KUKA KRL program: EPS_2_25862_MH6A_A_20251016034303.src

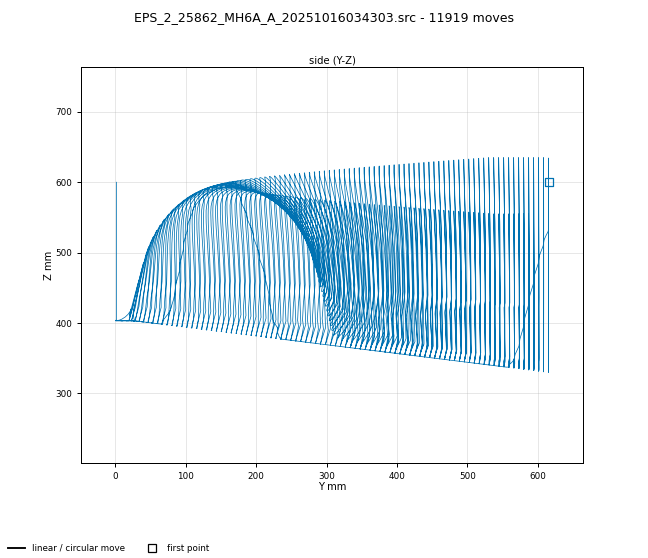
[picture p0: tool path of EPS_2_25862_MH6A_A_20251016034303.src, 11919 of 11921 moves have a stored position in this frame; points joined in program order, loops and branches not executed]
&ACCESS RVP
&REL 4
&COMMENT QRS 19112012
&PARAM EDITMASK = *
DEF PART()
EXT BAS (BAS_COMMAND :IN,REAL :IN )
INT I
BAS (#INITMOV,0 )

;KUKA QRS Post kuka4.cps  Date:22-06-2017 !

File_ID=2890

QRS_PRE_INIT()

;Init var - Until changes are made in qrs_pre_init
Outlet_Square_prg=0
Inlet_1_Square_prg=0
Inlet_2_Square_prg=0
Inlet_3_Square_prg=0
Inlet_4_Square_prg=0
Inlet_5_Square_prg=0

Outlet_1={X 0.000, Y 530.070, Z 534.500, B 0.000, E1 0.000 }
Inlet_1={X 0.000, Y 535.780, Z 454.500, B 0.000, E1 90.000 }
Outlet_1_type=201
Inlet_1_type=201
;QRS#1=Sidecore dimensions
;QRS#2=200-8" PVC SDR 35
;QRS#3=200-8" PVC SDR 35
;QRS#4=
;QRS#5=
;QRS#6=
;QRS#7=
;QRS#8=
;QRS#9=12-08 PSX
;QRS#10=12-08 PSX
;QRS#11=
;QRS#12=
;QRS#13=
;QRS#14=
;QRS#15=
;QRS#16=1220x127x914 3'
;QRS#17=EPS Height
;QRS#18=635
;QRS#19=*
;QRS#20= UPDATED VERSION 22-06-2017
;QRS#21=*
Outlet_Square=0100
Inlet_1_Square=0100
Inlet_2_Square=0
Inlet_3_Square=0
Inlet_4_Square=0
Inlet_5_Square=0
Mill_Square=1
Outlet_Square_Prg=204
Inlet_1_Square_prg=204

QRS_INIT()

$ADVANCE=5

; T1
PTP {E1 173.497,E2 173.497}
PTP {X 0,Y 615.499,A -85,B 0,C 180,E1 173.497,E2 173.497,E3 0,E4 0,E5 0,E6 0}
QRS_SPEED_INIT()
LIN {X 0,Y 615.499,Z 600,A -85,B 0,C 180,E1 173.497,E2 173.497,E3 0,E4 0,E5 0,E6 0} C_VEL
LIN {X 0,Y 615.499,Z 545.726,A -85,B 0,C 180,E1 173.497,E2 173.497} C_VEL
LIN {X 0,Y 615.499,Z 534.845,A -85,B 0,C 180,E1 173.497,E2 173.497} C_VEL
LIN {X 0,Y 615.497,Z 533.201,A -85,B 0,C 180,E1 173.417,E2 173.417} C_VEL
LIN {X 0,Y 615.497,Z 525.537,A -85,B 0,C 180,E1 172.455,E2 172.455} C_VEL
LIN {X 0,Y 615.498,Z 515.759,A -85,B 0,C 180,E1 171.464,E2 171.464} C_VEL
LIN {X 0,Y 615.497,Z 505.494,A -85,B 0,C 180,E1 170.636,E2 170.636} C_VEL
LIN {X 0,Y 615.479,Z 493.933,A -85,B 0,C 180,E1 169.889,E2 169.889} C_VEL
LIN {X 0,Y 615.498,Z 482.051,A -85,B 0,C 180,E1 169.292,E2 169.292} C_VEL
LIN {X 0,Y 615.49,Z 469.16,A -85,B 0,C 180,E1 168.807,E2 168.807} C_VEL
LIN {X 0,Y 615.493,Z 456.56,A -85,B 0,C 180,E1 168.473,E2 168.473} C_VEL
LIN {X 0,Y 615.494,Z 443.437,A -85,B 0,C 180,E1 168.265,E2 168.265} C_VEL
LIN {X 0,Y 615.492,Z 345.168,A -85,B 0,C 180,E1 167.114,E2 167.114} C_VEL
LIN {X 0,Y 615.479,Z 330.504,A -85,B 0,C 180,E1 164.265,E2 164.265} C_VEL
LIN {X 0,Y 615.477,Z 329.689,A -85,B 0,C 180,E1 164.095,E2 164.095} C_VEL
LIN {X 0,Y 615.484,Z 329.685,A -85,B 0,C 180,E1 161.354,E2 161.354} C_VEL
LIN {X 0,Y 615.494,Z 329.697,A -85,B 0,C 180,E1 158.568,E2 158.568} C_VEL
LIN {X 0,Y 615.488,Z 329.682,A -85,B 0,C 180,E1 155.728,E2 155.728} C_VEL
LIN {X 0,Y 615.488,Z 329.7,A -85,B 0,C 180,E1 152.823,E2 152.823} C_VEL
LIN {X 0,Y 615.477,Z 329.688,A -85,B 0,C 180,E1 150.208,E2 150.208} C_VEL
LIN {X 0,Y 615.491,Z 329.683,A -85,B 0,C 180,E1 147.543,E2 147.543} C_VEL
LIN {X 0,Y 615.483,Z 329.692,A -85,B 0,C 180,E1 145.185,E2 145.185} C_VEL
LIN {X 0,Y 615.495,Z 329.697,A -85,B 0,C 180,E1 142.758,E2 142.758} C_VEL
LIN {X 0,Y 615.486,Z 329.683,A -85,B 0,C 180,E1 139.912,E2 139.912} C_VEL
LIN {X 0,Y 615.494,Z 329.682,A -85,B 0,C 180,E1 137.648,E2 137.648} C_VEL
LIN {X 0,Y 615.497,Z 329.7,A -85,B 0,C 180,E1 134.932,E2 134.932} C_VEL
LIN {X 0,Y 615.479,Z 329.684,A -85,B 0,C 180,E1 132.079,E2 132.079} C_VEL
LIN {X 0,Y 615.495,Z 329.682,A -85,B 0,C 180,E1 129.75,E2 129.75} C_VEL
LIN {X 0,Y 615.494,Z 329.697,A -85,B 0,C 180,E1 126.937,E2 126.937} C_VEL
LIN {X 0,Y 615.482,Z 329.683,A -85,B 0,C 180,E1 124.023,E2 124.023} C_VEL
LIN {X 0,Y 615.492,Z 329.701,A -85,B 0,C 180,E1 121.086,E2 121.086} C_VEL
LIN {X 0,Y 615.477,Z 329.686,A -85,B 0,C 180,E1 118.448,E2 118.448} C_VEL
LIN {X 0,Y 615.493,Z 329.685,A -85,B 0,C 180,E1 115.716,E2 115.716} C_VEL
LIN {X 0,Y 615.49,Z 329.69,A -85,B 0,C 180,E1 112.845,E2 112.845} C_VEL
LIN {X 0,Y 615.483,Z 329.684,A -85,B 0,C 180,E1 110.034,E2 110.034} C_VEL
LIN {X 0,Y 615.497,Z 329.701,A -85,B 0,C 180,E1 107.271,E2 107.271} C_VEL
LIN {X 0,Y 615.479,Z 329.686,A -85,B 0,C 180,E1 104.55,E2 104.55} C_VEL
LIN {X 0,Y 615.49,Z 329.686,A -85,B 0,C 180,E1 101.861,E2 101.861} C_VEL
LIN {X 0,Y 615.496,Z 329.695,A -85,B 0,C 180,E1 99.199,E2 99.199} C_VEL
LIN {X 0,Y 615.478,Z 329.685,A -85,B 0,C 180,E1 96.557,E2 96.557} C_VEL
LIN {X 0,Y 615.491,Z 329.686,A -85,B 0,C 180,E1 93.929,E2 93.929} C_VEL
LIN {X 0,Y 615.496,Z 329.696,A -85,B 0,C 180,E1 91.309,E2 91.309} C_VEL
LIN {X 0,Y 615.48,Z 329.685,A -85,B 0,C 180,E1 88.692,E2 88.692} C_VEL
LIN {X 0,Y 615.489,Z 329.686,A -85,B 0,C 180,E1 86.072,E2 86.072} C_VEL
LIN {X 0,Y 615.496,Z 329.696,A -85,B 0,C 180,E1 83.416,E2 83.416} C_VEL
LIN {X 0,Y 615.48,Z 329.685,A -85,B 0,C 180,E1 80.802,E2 80.802} C_VEL
LIN {X 0,Y 615.488,Z 329.687,A -85,B 0,C 180,E1 78.14,E2 78.14} C_VEL
LIN {X 0,Y 615.494,Z 329.695,A -85,B 0,C 180,E1 75.452,E2 75.452} C_VEL
LIN {X 0,Y 615.478,Z 329.685,A -85,B 0,C 180,E1 72.73,E2 72.73} C_VEL
LIN {X 0,Y 615.494,Z 329.692,A -85,B 0,C 180,E1 69.968,E2 69.968} C_VEL
LIN {X 0,Y 615.49,Z 329.686,A -85,B 0,C 180,E1 67.157,E2 67.157} C_VEL
LIN {X 0,Y 615.489,Z 329.686,A -85,B 0,C 180,E1 64.285,E2 64.285} C_VEL
LIN {X 0,Y 615.491,Z 329.688,A -85,B 0,C 180,E1 61.343,E2 61.343} C_VEL
LIN {X 0,Y 615.482,Z 329.684,A -85,B 0,C 180,E1 58.915,E2 58.915} C_VEL
LIN {X 0,Y 615.482,Z 329.686,A -85,B 0,C 180,E1 56.467,E2 56.467} C_VEL
LIN {X 0,Y 615.493,Z 329.691,A -85,B 0,C 180,E1 54.166,E2 54.166} C_VEL
LIN {X 0,Y 615.496,Z 329.699,A -85,B 0,C 180,E1 51.933,E2 51.933} C_VEL
LIN {X 0,Y 615.487,Z 329.687,A -85,B 0,C 180,E1 49.395,E2 49.395} C_VEL
LIN {X 0,Y 615.476,Z 329.685,A -85,B 0,C 180,E1 46.756,E2 46.756} C_VEL
LIN {X 0,Y 615.491,Z 329.701,A -85,B 0,C 180,E1 43.999,E2 43.999} C_VEL
LIN {X 0,Y 615.49,Z 329.686,A -85,B 0,C 180,E1 41.474,E2 41.474} C_VEL
LIN {X 0,Y 615.478,Z 329.685,A -85,B 0,C 180,E1 38.905,E2 38.905} C_VEL
LIN {X 0,Y 615.488,Z 329.691,A -85,B 0,C 180,E1 36.425,E2 36.425} C_VEL
LIN {X 0,Y 615.489,Z 329.686,A -85,B 0,C 180,E1 33.536,E2 33.536} C_VEL
LIN {X 0,Y 615.478,Z 329.685,A -85,B 0,C 180,E1 30.92,E2 30.92} C_VEL
LIN {X 0,Y 615.491,Z 329.692,A -85,B 0,C 180,E1 28.453,E2 28.453} C_VEL
LIN {X 0,Y 615.488,Z 329.685,A -85,B 0,C 180,E1 25.572,E2 25.572} C_VEL
LIN {X 0,Y 615.475,Z 329.688,A -85,B 0,C 180,E1 22.845,E2 22.845} C_VEL
LIN {X 0,Y 615.487,Z 329.695,A -85,B 0,C 180,E1 20.033,E2 20.033} C_VEL
LIN {X 0,Y 615.489,Z 329.682,A -85,B 0,C 180,E1 17.27,E2 17.27} C_VEL
LIN {X 0,Y 615.49,Z 329.694,A -85,B 0,C 180,E1 14.549,E2 14.549} C_VEL
LIN {X 0,Y 615.481,Z 329.689,A -85,B 0,C 180,E1 11.861,E2 11.861} C_VEL
LIN {X 0,Y 615.483,Z 329.684,A -85,B 0,C 180,E1 9.199,E2 9.199} C_VEL
LIN {X 0,Y 615.492,Z 329.696,A -85,B 0,C 180,E1 6.557,E2 6.557} C_VEL
LIN {X 0,Y 615.476,Z 329.69,A -85,B 0,C 180,E1 3.929,E2 3.929} C_VEL
LIN {X 0,Y 615.486,Z 329.683,A -85,B 0,C 180,E1 1.309,E2 1.309} C_VEL
LIN {X 0,Y 615.485,Z 329.696,A -85,B 0,C 180,E1 -1.309,E2 -1.309} C_VEL
LIN {X 0,Y 615.476,Z 329.691,A -85,B 0,C 180,E1 -3.929,E2 -3.929} C_VEL
LIN {X 0,Y 615.49,Z 329.682,A -85,B 0,C 180,E1 -6.59,E2 -6.59} C_VEL
LIN {X 0,Y 615.483,Z 329.696,A -85,B 0,C 180,E1 -9.199,E2 -9.199} C_VEL
LIN {X 0,Y 615.478,Z 329.69,A -85,B 0,C 180,E1 -11.861,E2 -11.861} C_VEL
LIN {X 0,Y 615.49,Z 329.682,A -85,B 0,C 180,E1 -14.549,E2 -14.549} C_VEL
LIN {X 0,Y 615.495,Z 329.699,A -85,B 0,C 180,E1 -17.27,E2 -17.27} C_VEL
LIN {X 0,Y 615.479,Z 329.686,A -85,B 0,C 180,E1 -20.033,E2 -20.033} C_VEL
LIN {X 0,Y 615.482,Z 329.69,A -85,B 0,C 180,E1 -22.845,E2 -22.845} C_VEL
LIN {X 0,Y 615.485,Z 329.692,A -85,B 0,C 180,E1 -25.571,E2 -25.571} C_VEL
LIN {X 0,Y 615.492,Z 329.682,A -85,B 0,C 180,E1 -28.454,E2 -28.454} C_VEL
LIN {X 0,Y 615.487,Z 329.7,A -85,B 0,C 180,E1 -31.088,E2 -31.088} C_VEL
LIN {X 0,Y 615.484,Z 329.691,A -85,B 0,C 180,E1 -33.536,E2 -33.536} C_VEL
LIN {X 0,Y 615.489,Z 329.684,A -85,B 0,C 180,E1 -36.425,E2 -36.425} C_VEL
LIN {X 0,Y 615.496,Z 329.7,A -85,B 0,C 180,E1 -39.065,E2 -39.065} C_VEL
LIN {X 0,Y 615.485,Z 329.69,A -85,B 0,C 180,E1 -41.474,E2 -41.474} C_VEL
LIN {X 0,Y 615.491,Z 329.682,A -85,B 0,C 180,E1 -44.149,E2 -44.149} C_VEL
LIN {X 0,Y 615.492,Z 329.7,A -85,B 0,C 180,E1 -46.952,E2 -46.952} C_VEL
LIN {X 0,Y 615.483,Z 329.69,A -85,B 0,C 180,E1 -49.395,E2 -49.395} C_VEL
LIN {X 0,Y 615.484,Z 329.683,A -85,B 0,C 180,E1 -51.989,E2 -51.989} C_VEL
LIN {X 0,Y 615.491,Z 329.686,A -85,B 0,C 180,E1 -54.386,E2 -54.386} C_VEL
LIN {X 0,Y 615.487,Z 329.698,A -85,B 0,C 180,E1 -56.765,E2 -56.765} C_VEL
LIN {X 0,Y 615.496,Z 329.693,A -85,B 0,C 180,E1 -59.082,E2 -59.082} C_VEL
LIN {X 0,Y 615.477,Z 329.686,A -85,B 0,C 180,E1 -61.552,E2 -61.552} C_VEL
LIN {X 0,Y 615.493,Z 329.686,A -85,B 0,C 180,E1 -64.286,E2 -64.286} C_VEL
LIN {X 0,Y 615.483,Z 329.765,A -85,B 0,C 180,E1 -66.022,E2 -66.022} C_VEL
LIN {X 0,Y 615.486,Z 351.817,A -85,B 0,C 180,E1 -68.745,E2 -68.745} C_VEL
LIN {X 0,Y 615.494,Z 375,A -85,B 0,C 180,E1 -71.556,E2 -71.556} C_VEL
LIN {X 0,Y 615.486,Z 397.682,A -85,B 0,C 180,E1 -74.266,E2 -74.266} C_VEL
LIN {X 0,Y 615.498,Z 421.822,A -85,B 0,C 180,E1 -77.115,E2 -77.115} C_VEL
LIN {X 0,Y 615.479,Z 530.88,A -85,B 0,C 180,E1 -78.411,E2 -78.411} C_VEL
LIN {X 0,Y 615.478,Z 543.377,A -85,B 0,C 180,E1 -78.683,E2 -78.683} C_VEL
LIN {X 0,Y 615.491,Z 556.57,A -85,B 0,C 180,E1 -79.111,E2 -79.111} C_VEL
LIN {X 0,Y 615.478,Z 568.495,A -85,B 0,C 180,E1 -79.64,E2 -79.64} C_VEL
LIN {X 0,Y 615.487,Z 580.008,A -85,B 0,C 180,E1 -80.305,E2 -80.305} C_VEL
LIN {X 0,Y 615.499,Z 590.352,A -85,B 0,C 180,E1 -81.051,E2 -81.051} C_VEL
LIN {X 0,Y 615.497,Z 598.82,A -85,B 0,C 180,E1 -81.795,E2 -81.795} C_VEL
LIN {X 0,Y 615.497,Z 607.972,A -85,B 0,C 180,E1 -82.785,E2 -82.785} C_VEL
LIN {X 0,Y 615.497,Z 615.321,A -85,B 0,C 180,E1 -83.773,E2 -83.773} C_VEL
LIN {X 0,Y 615.499,Z 621.209,A -85,B 0,C 180,E1 -84.76,E2 -84.76} C_VEL
LIN {X 0,Y 615.493,Z 625.855,A -85,B 0,C 180,E1 -85.744,E2 -85.744} C_VEL
LIN {X 0,Y 615.495,Z 629.401,A -85,B 0,C 180,E1 -86.728,E2 -86.728} C_VEL
LIN {X 0,Y 615.497,Z 631.235,A -85,B 0,C 180,E1 -87.383,E2 -87.383} C_VEL
LIN {X 0,Y 615.497,Z 632.609,A -85,B 0,C 180,E1 -88.038,E2 -88.038} C_VEL
LIN {X 0,Y 615.496,Z 634.174,A -85,B 0,C 180,E1 -89.347,E2 -89.347} C_VEL
LIN {X 0,Y 615.494,Z 634.389,A -85,B 0,C 180,E1 -90.001,E2 -90.001} C_VEL
LIN {X 0,Y 615.496,Z 633.579,A -85,B 0,C 180,E1 -91.309,E2 -91.309} C_VEL
LIN {X 0,Y 615.497,Z 632.607,A -85,B 0,C 180,E1 -91.964,E2 -91.964} C_VEL
LIN {X 0,Y 615.497,Z 631.231,A -85,B 0,C 180,E1 -92.619,E2 -92.619} C_VEL
LIN {X 0,Y 615.496,Z 628.347,A -85,B 0,C 180,E1 -93.601,E2 -93.601} C_VEL
LIN {X 0,Y 615.498,Z 624.438,A -85,B 0,C 180,E1 -94.585,E2 -94.585} C_VEL
LIN {X 0,Y 615.499,Z 619.401,A -85,B 0,C 180,E1 -95.57,E2 -95.57} C_VEL
LIN {X 0,Y 615.497,Z 612.87,A -85,B 0,C 180,E1 -96.583,E2 -96.583} C_VEL
LIN {X 0,Y 615.497,Z 605.127,A -85,B 0,C 180,E1 -97.546,E2 -97.546} C_VEL
LIN {X 0,Y 615.498,Z 597.037,A -85,B 0,C 180,E1 -98.372,E2 -98.372} C_VEL
LIN {X 0,Y 615.499,Z 587.158,A -85,B 0,C 180,E1 -99.199,E2 -99.199} C_VEL
LIN {X 0,Y 615.488,Z 575.97,A -85,B 0,C 180,E1 -99.946,E2 -99.946} C_VEL
LIN {X 0,Y 615.481,Z 565.009,A -85,B 0,C 180,E1 -100.528,E2 -100.528} C_VEL
LIN {X 0,Y 615.49,Z 552.439,A -85,B 0,C 180,E1 -101.042,E2 -101.042} C_VEL
LIN {X 0,Y 615.477,Z 540.037,A -85,B 0,C 180,E1 -101.402,E2 -101.402} C_VEL
LIN {X 0,Y 615.481,Z 526.418,A -85,B 0,C 180,E1 -101.653,E2 -101.653} C_VEL
LIN {X 0,Y 615.498,Z 421.809,A -85,B 0,C 180,E1 -102.887,E2 -102.887} C_VEL
LIN {X 0,Y 615.486,Z 397.669,A -85,B 0,C 180,E1 -105.736,E2 -105.736} C_VEL
LIN {X 0,Y 615.498,Z 373.644,A -85,B 0,C 180,E1 -108.607,E2 -108.607} C_VEL
LIN {X 0,Y 615.488,Z 350.368,A -85,B 0,C 180,E1 -111.432,E2 -111.432} C_VEL
LIN {X 0,Y 615.486,Z 329.684,A -85,B 0,C 180,E1 -114.007,E2 -114.007} C_VEL
LIN {X 0,Y 615.478,Z 329.686,A -85,B 0,C 180,E1 -116.445,E2 -116.445} C_VEL
LIN {X 0,Y 615.485,Z 329.688,A -85,B 0,C 180,E1 -118.659,E2 -118.659} C_VEL
LIN {X 0,Y 615.495,Z 329.699,A -85,B 0,C 180,E1 -121.087,E2 -121.087} C_VEL
LIN {X 0,Y 615.483,Z 329.683,A -85,B 0,C 180,E1 -124.023,E2 -124.023} C_VEL
LIN {X 0,Y 615.494,Z 329.696,A -85,B 0,C 180,E1 -126.937,E2 -126.937} C_VEL
LIN {X 0,Y 615.495,Z 329.682,A -85,B 0,C 180,E1 -129.75,E2 -129.75} C_VEL
LIN {X 0,Y 615.476,Z 329.687,A -85,B 0,C 180,E1 -132.355,E2 -132.355} C_VEL
LIN {X 0,Y 615.493,Z 329.699,A -85,B 0,C 180,E1 -135.069,E2 -135.069} C_VEL
LIN {X 0,Y 615.486,Z 329.683,A -85,B 0,C 180,E1 -137.921,E2 -137.921} C_VEL
LIN {X 0,Y 615.477,Z 329.686,A -85,B 0,C 180,E1 -140.249,E2 -140.249} C_VEL
LIN {X 0,Y 615.492,Z 329.697,A -85,B 0,C 180,E1 -143.064,E2 -143.064} C_VEL
LIN {X 0,Y 615.481,Z 329.684,A -85,B 0,C 180,E1 -145.977,E2 -145.977} C_VEL
LIN {X 0,Y 615.479,Z 329.688,A -85,B 0,C 180,E1 -148.314,E2 -148.314} C_VEL
LIN {X 0,Y 615.489,Z 329.693,A -85,B 0,C 180,E1 -150.594,E2 -150.594} C_VEL
LIN {X 0,Y 615.494,Z 329.682,A -85,B 0,C 180,E1 -153.556,E2 -153.556} C_VEL
LIN {X 0,Y 615.485,Z 329.691,A -85,B 0,C 180,E1 -156.443,E2 -156.443} C_VEL
LIN {X 0,Y 615.484,Z 329.688,A -85,B 0,C 180,E1 -159.269,E2 -159.269} C_VEL
LIN {X 0,Y 615.477,Z 329.686,A -85,B 0,C 180,E1 -162.043,E2 -162.043} C_VEL
LIN {X 0,Y 615.478,Z 329.826,A -85,B 0,C 180,E1 -164.222,E2 -164.222} C_VEL
LIN {X 0,Y 615.495,Z 343.07,A -85,B 0,C 180,E1 -166.799,E2 -166.799} C_VEL
LIN {X 0,Y 615.494,Z 345.135,A -85,B 0,C 180,E1 -167.197,E2 -167.197} C_VEL
LIN {X 0,Y 615.494,Z 450.636,A -85,B 0,C 180,E1 -168.452,E2 -168.452} C_VEL
LIN {X 0,Y 615.491,Z 463.219,A -85,B 0,C 180,E1 -168.724,E2 -168.724} C_VEL
LIN {X 0,Y 615.491,Z 476.604,A -85,B 0,C 180,E1 -169.158,E2 -169.158} C_VEL
LIN {X 0,Y 615.492,Z 487.563,A -85,B 0,C 180,E1 -169.639,E2 -169.639} C_VEL
LIN {X 0,Y 615.482,Z 499.304,A -85,B 0,C 180,E1 -170.304,E2 -170.304} C_VEL
LIN {X 0,Y 615.499,Z 509.766,A -85,B 0,C 180,E1 -171.05,E2 -171.05} C_VEL
LIN {X 0,Y 615.498,Z 518.329,A -85,B 0,C 180,E1 -171.794,E2 -171.794} C_VEL
LIN {X 0,Y 615.498,Z 526.208,A -85,B 0,C 180,E1 -172.619,E2 -172.619} C_VEL
LIN {X 0,Y 615.497,Z 533.898,A -85,B 0,C 180,E1 -173.608,E2 -173.608} C_VEL
LIN {X 0,Y 615.498,Z 540.957,A -85,B 0,C 180,E1 -174.759,E2 -174.759} C_VEL
LIN {X 0,Y 615.493,Z 545.657,A -85,B 0,C 180,E1 -175.744,E2 -175.744} C_VEL
LIN {X 0,Y 615.496,Z 549.254,A -85,B 0,C 180,E1 -176.727,E2 -176.727} C_VEL
LIN {X 0,Y 615.496,Z 551.114,A -85,B 0,C 180,E1 -177.382,E2 -177.382} C_VEL
LIN {X 0,Y 615.497,Z 552.533,A -85,B 0,C 180,E1 -178.037,E2 -178.037} C_VEL
LIN {X 0,Y 615.496,Z 554.141,A -85,B 0,C 180,E1 -179.346,E2 -179.346} C_VEL
LIN {X 0,Y 615.494,Z 554.384,A -85,B 0,C 180,E1 -180,E2 -180} C_VEL
LIN {X 0,Y 615.496,Z 554.206,A -85,B 0,C 180,E1 -180.654,E2 -180.654} C_VEL
LIN {X 0,Y 615.496,Z 552.683,A -85,B 0,C 180,E1 -181.963,E2 -181.963} C_VEL
LIN {X 0,Y 615.498,Z 551.341,A -85,B 0,C 180,E1 -182.618,E2 -182.618} C_VEL
LIN {X 0,Y 615.497,Z 548.494,A -85,B 0,C 180,E1 -183.601,E2 -183.601} C_VEL
LIN {X 0,Y 615.499,Z 544.634,A -85,B 0,C 180,E1 -184.584,E2 -184.584} C_VEL
LIN {X 0,Y 615.498,Z 539.652,A -85,B 0,C 180,E1 -185.57,E2 -185.57} C_VEL
LIN {X 0,Y 615.497,Z 533.201,A -85,B 0,C 180,E1 -186.583,E2 -186.583} C_VEL
LIN {X 0,Y 614.829,Z 530.019,A -85,B 0,C 180,E1 -187.032,E2 -187.032} C_VEL
LIN {X 0,Y 611.988,Z 524.446,A -85,B 0,C 180,E1 -187.749,E2 -187.749} C_VEL
LIN {X 0,Y 609.138,Z 518.17,A -85,B 0,C 180,E1 -188.43,E2 -188.43} C_VEL
LIN {X 0,Y 608.477,Z 513.929,A -85,B 0,C 180,E1 -188.82,E2 -188.82} C_VEL
LIN {X 0,Y 608.489,Z 503.393,A -85,B 0,C 180,E1 -189.641,E2 -189.641} C_VEL
LIN {X 0,Y 608.49,Z 492.613,A -85,B 0,C 180,E1 -190.313,E2 -190.313} C_VEL
LIN {X 0,Y 608.522,Z 479.878,A -85,B 0,C 180,E1 -190.931,E2 -190.931} C_VEL
LIN {X 0,Y 608.523,Z 467.972,A -85,B 0,C 180,E1 -191.365,E2 -191.365} C_VEL
LIN {X 0,Y 608.554,Z 455.647,A -85,B 0,C 180,E1 -191.681,E2 -191.681} C_VEL
LIN {X 0,Y 608.556,Z 441.756,A -85,B 0,C 180,E1 -191.892,E2 -191.892} C_VEL
LIN {X 0,Y 608.474,Z 345.388,A -85,B 0,C 180,E1 -193.038,E2 -193.038} C_VEL
LIN {X 0,Y 608.469,Z 330.765,A -85,B 0,C 180,E1 -195.9,E2 -195.9} C_VEL
LIN {X 0,Y 608.457,Z 330.69,A -85,B 0,C 180,E1 -198.87,E2 -198.87} C_VEL
LIN {X 0,Y 608.471,Z 330.689,A -85,B 0,C 180,E1 -201.691,E2 -201.691} C_VEL
LIN {X 0,Y 608.455,Z 330.688,A -85,B 0,C 180,E1 -204.571,E2 -204.571} C_VEL
LIN {X 0,Y 608.482,Z 330.694,A -85,B 0,C 180,E1 -207.207,E2 -207.207} C_VEL
LIN {X 0,Y 608.463,Z 330.687,A -85,B 0,C 180,E1 -209.97,E2 -209.97} C_VEL
LIN {X 0,Y 608.463,Z 330.692,A -85,B 0,C 180,E1 -212.879,E2 -212.879} C_VEL
LIN {X 0,Y 608.439,Z 330.698,A -85,B 0,C 180,E1 -215.278,E2 -215.278} C_VEL
LIN {X 0,Y 608.47,Z 330.687,A -85,B 0,C 180,E1 -217.746,E2 -217.746} C_VEL
LIN {X 0,Y 608.451,Z 330.688,A -85,B 0,C 180,E1 -220.328,E2 -220.328} C_VEL
LIN {X 0,Y 608.485,Z 330.69,A -85,B 0,C 180,E1 -223.31,E2 -223.31} C_VEL
LIN {X 0,Y 608.469,Z 330.685,A -85,B 0,C 180,E1 -226.13,E2 -226.13} C_VEL
LIN {X 0,Y 608.461,Z 330.694,A -85,B 0,C 180,E1 -228.823,E2 -228.823} C_VEL
LIN {X 0,Y 608.474,Z 330.688,A -85,B 0,C 180,E1 -231.412,E2 -231.412} C_VEL
LIN {X 0,Y 608.45,Z 330.688,A -85,B 0,C 180,E1 -233.954,E2 -233.954} C_VEL
LIN {X 0,Y 608.452,Z 330.689,A -85,B 0,C 180,E1 -236.328,E2 -236.328} C_VEL
LIN {X 0,Y 608.483,Z 330.691,A -85,B 0,C 180,E1 -238.727,E2 -238.727} C_VEL
LIN {X 0,Y 608.47,Z 330.688,A -85,B 0,C 180,E1 -241.381,E2 -241.381} C_VEL
LIN {X 0,Y 608.446,Z 330.688,A -85,B 0,C 180,E1 -243.964,E2 -243.964} C_VEL
LIN {X 0,Y 608.466,Z 330.687,A -85,B 0,C 180,E1 -246.154,E2 -246.154} C_VEL
LIN {X 0,Y 608.458,Z 330.693,A -85,B 0,C 180,E1 -249.018,E2 -249.018} C_VEL
LIN {X 0,Y 608.454,Z 330.687,A -85,B 0,C 180,E1 -251.828,E2 -251.828} C_VEL
LIN {X 0,Y 608.478,Z 330.693,A -85,B 0,C 180,E1 -254.594,E2 -254.594} C_VEL
LIN {X 0,Y 608.472,Z 330.686,A -85,B 0,C 180,E1 -257.322,E2 -257.322} C_VEL
LIN {X 0,Y 608.461,Z 330.688,A -85,B 0,C 180,E1 -260.022,E2 -260.022} C_VEL
LIN {X 0,Y 608.489,Z 330.692,A -85,B 0,C 180,E1 -262.7,E2 -262.7} C_VEL
LIN {X 0,Y 608.448,Z 330.688,A -85,B 0,C 180,E1 -265.362,E2 -265.362} C_VEL
LIN {X 0,Y 608.468,Z 330.688,A -85,B 0,C 180,E1 -268.014,E2 -268.014} C_VEL
LIN {X 0,Y 608.487,Z 330.691,A -85,B 0,C 180,E1 -270.661,E2 -270.661} C_VEL
LIN {X 0,Y 608.475,Z 330.685,A -85,B 0,C 180,E1 -273.31,E2 -273.31} C_VEL
LIN {X 0,Y 608.49,Z 330.685,A -85,B 0,C 180,E1 -275.966,E2 -275.966} C_VEL
LIN {X 0,Y 608.461,Z 330.694,A -85,B 0,C 180,E1 -278.635,E2 -278.635} C_VEL
LIN {X 0,Y 608.475,Z 330.685,A -85,B 0,C 180,E1 -281.323,E2 -281.323} C_VEL
LIN {X 0,Y 608.471,Z 330.69,A -85,B 0,C 180,E1 -284.037,E2 -284.037} C_VEL
LIN {X 0,Y 608.477,Z 330.688,A -85,B 0,C 180,E1 -286.782,E2 -286.782} C_VEL
LIN {X 0,Y 608.448,Z 330.689,A -85,B 0,C 180,E1 -289.57,E2 -289.57} C_VEL
LIN {X 0,Y 608.475,Z 330.693,A -85,B 0,C 180,E1 -292.404,E2 -292.404} C_VEL
LIN {X 0,Y 608.457,Z 330.692,A -85,B 0,C 180,E1 -294.57,E2 -294.57} C_VEL
LIN {X 0,Y 608.475,Z 330.684,A -85,B 0,C 180,E1 -297.206,E2 -297.206} C_VEL
LIN {X 0,Y 608.477,Z 330.691,A -85,B 0,C 180,E1 -299.973,E2 -299.973} C_VEL
LIN {X 0,Y 608.464,Z 330.691,A -85,B 0,C 180,E1 -302.523,E2 -302.523} C_VEL
LIN {X 0,Y 608.447,Z 330.688,A -85,B 0,C 180,E1 -305.276,E2 -305.276} C_VEL
LIN {X 0,Y 608.474,Z 330.693,A -85,B 0,C 180,E1 -308.241,E2 -308.241} C_VEL
LIN {X 0,Y 608.477,Z 330.691,A -85,B 0,C 180,E1 -310.332,E2 -310.332} C_VEL
LIN {X 0,Y 608.449,Z 330.688,A -85,B 0,C 180,E1 -312.959,E2 -312.959} C_VEL
LIN {X 0,Y 608.462,Z 330.692,A -85,B 0,C 180,E1 -315.734,E2 -315.734} C_VEL
LIN {X 0,Y 608.462,Z 330.687,A -85,B 0,C 180,E1 -318.656,E2 -318.656} C_VEL
LIN {X 0,Y 608.466,Z 330.688,A -85,B 0,C 180,E1 -321.412,E2 -321.412} C_VEL
LIN {X 0,Y 608.472,Z 330.696,A -85,B 0,C 180,E1 -323.949,E2 -323.949} C_VEL
LIN {X 0,Y 608.468,Z 330.689,A -85,B 0,C 180,E1 -326.33,E2 -326.33} C_VEL
LIN {X 0,Y 608.471,Z 330.685,A -85,B 0,C 180,E1 -328.726,E2 -328.726} C_VEL
LIN {X 0,Y 608.471,Z 330.688,A -85,B 0,C 180,E1 -331.378,E2 -331.378} C_VEL
LIN {X 0,Y 608.469,Z 330.688,A -85,B 0,C 180,E1 -334.277,E2 -334.277} C_VEL
LIN {X 0,Y 608.445,Z 330.688,A -85,B 0,C 180,E1 -336.876,E2 -336.876} C_VEL
LIN {X 0,Y 608.464,Z 330.689,A -85,B 0,C 180,E1 -339.319,E2 -339.319} C_VEL
LIN {X 0,Y 608.447,Z 330.697,A -85,B 0,C 180,E1 -341.828,E2 -341.828} C_VEL
LIN {X 0,Y 608.468,Z 330.685,A -85,B 0,C 180,E1 -344.594,E2 -344.594} C_VEL
LIN {X 0,Y 608.474,Z 330.689,A -85,B 0,C 180,E1 -347.323,E2 -347.323} C_VEL
LIN {X 0,Y 608.453,Z 330.691,A -85,B 0,C 180,E1 -350.023,E2 -350.023} C_VEL
LIN {X 0,Y 608.477,Z 330.684,A -85,B 0,C 180,E1 -352.701,E2 -352.701} C_VEL
LIN {X 0,Y 608.459,Z 330.693,A -85,B 0,C 180,E1 -355.362,E2 -355.362} C_VEL
LIN {X 0,Y 608.448,Z 330.691,A -85,B 0,C 180,E1 -358.014,E2 -358.014} C_VEL
LIN {X 0,Y 608.478,Z 330.684,A -85,B 0,C 180,E1 -360.662,E2 -360.662} C_VEL
LIN {X 0,Y 608.476,Z 330.692,A -85,B 0,C 180,E1 -363.311,E2 -363.311} C_VEL
LIN {X 0,Y 608.451,Z 330.69,A -85,B 0,C 180,E1 -365.967,E2 -365.967} C_VEL
LIN {X 0,Y 608.455,Z 330.687,A -85,B 0,C 180,E1 -368.636,E2 -368.636} C_VEL
LIN {X 0,Y 608.472,Z 330.694,A -85,B 0,C 180,E1 -371.324,E2 -371.324} C_VEL
LIN {X 0,Y 608.459,Z 330.688,A -85,B 0,C 180,E1 -374.038,E2 -374.038} C_VEL
LIN {X 0,Y 608.474,Z 330.687,A -85,B 0,C 180,E1 -376.784,E2 -376.784} C_VEL
LIN {X 0,Y 608.45,Z 330.694,A -85,B 0,C 180,E1 -379.571,E2 -379.571} C_VEL
LIN {X 0,Y 608.456,Z 330.687,A -85,B 0,C 180,E1 -382.478,E2 -382.478} C_VEL
LIN {X 0,Y 608.45,Z 330.698,A -85,B 0,C 180,E1 -385.301,E2 -385.301} C_VEL
LIN {X 0,Y 608.446,Z 330.693,A -85,B 0,C 180,E1 -387.518,E2 -387.518} C_VEL
LIN {X 0,Y 608.461,Z 330.687,A -85,B 0,C 180,E1 -389.973,E2 -389.973} C_VEL
LIN {X 0,Y 608.464,Z 330.687,A -85,B 0,C 180,E1 -392.525,E2 -392.525} C_VEL
LIN {X 0,Y 608.44,Z 330.697,A -85,B 0,C 180,E1 -395.278,E2 -395.278} C_VEL
LIN {X 0,Y 608.469,Z 330.687,A -85,B 0,C 180,E1 -397.746,E2 -397.746} C_VEL
LIN {X 0,Y 608.476,Z 330.685,A -85,B 0,C 180,E1 -400.333,E2 -400.333} C_VEL
LIN {X 0,Y 608.484,Z 330.689,A -85,B 0,C 180,E1 -403.312,E2 -403.312} C_VEL
LIN {X 0,Y 608.468,Z 330.686,A -85,B 0,C 180,E1 -406.132,E2 -406.132} C_VEL
LIN {X 0,Y 608.46,Z 330.694,A -85,B 0,C 180,E1 -408.825,E2 -408.825} C_VEL
LIN {X 0,Y 608.473,Z 330.688,A -85,B 0,C 180,E1 -411.414,E2 -411.414} C_VEL
LIN {X 0,Y 608.475,Z 330.684,A -85,B 0,C 180,E1 -413.951,E2 -413.951} C_VEL
LIN {X 0,Y 608.464,Z 330.688,A -85,B 0,C 180,E1 -416.331,E2 -416.331} C_VEL
LIN {X 0,Y 608.478,Z 330.692,A -85,B 0,C 180,E1 -418.728,E2 -418.728} C_VEL
LIN {X 0,Y 608.469,Z 330.688,A -85,B 0,C 180,E1 -421.381,E2 -421.381} C_VEL
LIN {X 0,Y 608.446,Z 330.689,A -85,B 0,C 180,E1 -423.966,E2 -423.966} C_VEL
LIN {X 0,Y 608.475,Z 330.722,A -85,B 0,C 180,E1 -425.849,E2 -425.849} C_VEL
LIN {X 0,Y 608.596,Z 344.642,A -85,B 0,C 180,E1 -427.6,E2 -427.6} C_VEL
LIN {X 0,Y 608.572,Z 366.167,A -85,B 0,C 180,E1 -430.259,E2 -430.259} C_VEL
LIN {X 0,Y 608.534,Z 389.127,A -85,B 0,C 180,E1 -433.046,E2 -433.046} C_VEL
LIN {X 0,Y 608.503,Z 412.087,A -85,B 0,C 180,E1 -435.794,E2 -435.794} C_VEL
LIN {X 0,Y 608.507,Z 421.953,A -85,B 0,C 180,E1 -436.964,E2 -436.964} C_VEL
LIN {X 0,Y 608.538,Z 530.994,A -85,B 0,C 180,E1 -438.277,E2 -438.277} C_VEL
LIN {X 0,Y 608.514,Z 544.248,A -85,B 0,C 180,E1 -438.572,E2 -438.572} C_VEL
LIN {X 0,Y 608.517,Z 556.604,A -85,B 0,C 180,E1 -438.981,E2 -438.981} C_VEL
LIN {X 0,Y 608.498,Z 568.651,A -85,B 0,C 180,E1 -439.52,E2 -439.52} C_VEL
LIN {X 0,Y 608.48,Z 580.21,A -85,B 0,C 180,E1 -440.192,E2 -440.192} C_VEL
LIN {X 0,Y 608.485,Z 590.604,A -85,B 0,C 180,E1 -440.947,E2 -440.947} C_VEL
LIN {X 0,Y 608.475,Z 599.121,A -85,B 0,C 180,E1 -441.7,E2 -441.7} C_VEL
LIN {X 0,Y 608.47,Z 606.967,A -85,B 0,C 180,E1 -442.535,E2 -442.535} C_VEL
LIN {X 0,Y 608.46,Z 614.29,A -85,B 0,C 180,E1 -443.485,E2 -443.485} C_VEL
LIN {X 0,Y 608.45,Z 619.87,A -85,B 0,C 180,E1 -444.366,E2 -444.366} C_VEL
LIN {X 0,Y 608.432,Z 624.953,A -85,B 0,C 180,E1 -445.363,E2 -445.363} C_VEL
LIN {X 0,Y 608.449,Z 628.899,A -85,B 0,C 180,E1 -446.358,E2 -446.358} C_VEL
LIN {X 0,Y 608.425,Z 631.811,A -85,B 0,C 180,E1 -447.353,E2 -447.353} C_VEL
LIN {X 0,Y 608.442,Z 633.203,A -85,B 0,C 180,E1 -448.015,E2 -448.015} C_VEL
LIN {X 0,Y 608.439,Z 634.784,A -85,B 0,C 180,E1 -449.339,E2 -449.339} C_VEL
LIN {X 0,Y 608.434,Z 635,A -85,B 0,C 180,E1 -450.001,E2 -450.001} C_VEL
LIN {X 0,Y 608.448,Z 634.183,A -85,B 0,C 180,E1 -451.324,E2 -451.324} C_VEL
LIN {X 0,Y 608.443,Z 633.2,A -85,B 0,C 180,E1 -451.987,E2 -451.987} C_VEL
LIN {X 0,Y 608.425,Z 631.807,A -85,B 0,C 180,E1 -452.649,E2 -452.649} C_VEL
LIN {X 0,Y 608.449,Z 628.894,A -85,B 0,C 180,E1 -453.643,E2 -453.643} C_VEL
LIN {X 0,Y 608.432,Z 624.947,A -85,B 0,C 180,E1 -454.639,E2 -454.639} C_VEL
LIN {X 0,Y 608.437,Z 618.872,A -85,B 0,C 180,E1 -455.802,E2 -455.802} C_VEL
LIN {X 0,Y 608.463,Z 612.23,A -85,B 0,C 180,E1 -456.8,E2 -456.8} C_VEL
LIN {X 0,Y 608.456,Z 603.983,A -85,B 0,C 180,E1 -457.801,E2 -457.801} C_VEL
LIN {X 0,Y 608.472,Z 595.528,A -85,B 0,C 180,E1 -458.637,E2 -458.637} C_VEL
LIN {X 0,Y 608.471,Z 585.081,A -85,B 0,C 180,E1 -459.474,E2 -459.474} C_VEL
LIN {X 0,Y 608.494,Z 574.744,A -85,B 0,C 180,E1 -460.145,E2 -460.145} C_VEL
LIN {X 0,Y 608.521,Z 563.24,A -85,B 0,C 180,E1 -460.741,E2 -460.741} C_VEL
LIN {X 0,Y 608.531,Z 550.863,A -85,B 0,C 180,E1 -461.226,E2 -461.226} C_VEL
LIN {X 0,Y 608.537,Z 537.409,A -85,B 0,C 180,E1 -461.598,E2 -461.598} C_VEL
LIN {X 0,Y 608.547,Z 525.03,A -85,B 0,C 180,E1 -461.809,E2 -461.809} C_VEL
LIN {X 0,Y 608.507,Z 421.94,A -85,B 0,C 180,E1 -463.038,E2 -463.038} C_VEL
LIN {X 0,Y 608.528,Z 397.724,A -85,B 0,C 180,E1 -465.921,E2 -465.921} C_VEL
LIN {X 0,Y 608.57,Z 373.329,A -85,B 0,C 180,E1 -468.867,E2 -468.867} C_VEL
LIN {X 0,Y 608.597,Z 350.368,A -85,B 0,C 180,E1 -471.687,E2 -471.687} C_VEL
LIN {X 0,Y 608.598,Z 331.358,A -85,B 0,C 180,E1 -474.066,E2 -474.066} C_VEL
LIN {X 0,Y 608.464,Z 330.688,A -85,B 0,C 180,E1 -474.196,E2 -474.196} C_VEL
LIN {X 0,Y 608.452,Z 330.691,A -85,B 0,C 180,E1 -476.775,E2 -476.775} C_VEL
LIN {X 0,Y 608.482,Z 330.685,A -85,B 0,C 180,E1 -479.779,E2 -479.779} C_VEL
LIN {X 0,Y 608.456,Z 330.689,A -85,B 0,C 180,E1 -482.521,E2 -482.521} C_VEL
LIN {X 0,Y 608.451,Z 330.695,A -85,B 0,C 180,E1 -485.278,E2 -485.278} C_VEL
LIN {X 0,Y 608.47,Z 330.686,A -85,B 0,C 180,E1 -487.747,E2 -487.747} C_VEL
LIN {X 0,Y 608.445,Z 330.689,A -85,B 0,C 180,E1 -490.328,E2 -490.328} C_VEL
LIN {X 0,Y 608.478,Z 330.69,A -85,B 0,C 180,E1 -493.309,E2 -493.309} C_VEL
LIN {X 0,Y 608.47,Z 330.685,A -85,B 0,C 180,E1 -496.13,E2 -496.13} C_VEL
LIN {X 0,Y 608.462,Z 330.694,A -85,B 0,C 180,E1 -498.824,E2 -498.824} C_VEL
LIN {X 0,Y 608.467,Z 330.686,A -85,B 0,C 180,E1 -501.76,E2 -501.76} C_VEL
LIN {X 0,Y 608.449,Z 330.688,A -85,B 0,C 180,E1 -503.955,E2 -503.955} C_VEL
LIN {X 0,Y 608.451,Z 330.69,A -85,B 0,C 180,E1 -506.328,E2 -506.328} C_VEL
LIN {X 0,Y 608.452,Z 330.696,A -85,B 0,C 180,E1 -508.732,E2 -508.732} C_VEL
LIN {X 0,Y 608.477,Z 330.687,A -85,B 0,C 180,E1 -511.38,E2 -511.38} C_VEL
LIN {X 0,Y 608.445,Z 330.688,A -85,B 0,C 180,E1 -513.964,E2 -513.964} C_VEL
LIN {X 0,Y 608.461,Z 330.688,A -85,B 0,C 180,E1 -516.155,E2 -516.155} C_VEL
LIN {X 0,Y 608.471,Z 330.688,A -85,B 0,C 180,E1 -518.308,E2 -518.308} C_VEL
LIN {X 0,Y 608.474,Z 330.687,A -85,B 0,C 180,E1 -521.284,E2 -521.284} C_VEL
LIN {X 0,Y 608.455,Z 330.744,A -85,B 0,C 180,E1 -524.186,E2 -524.186} C_VEL
LIN {X 0,Y 608.462,Z 345.033,A -85,B 0,C 180,E1 -526.983,E2 -526.983} C_VEL
LIN {X 0,Y 608.476,Z 345.6,A -85,B 0,C 180,E1 -527.058,E2 -527.058} C_VEL
LIN {X 0,Y 608.555,Z 450.792,A -85,B 0,C 180,E1 -528.319,E2 -528.319} C_VEL
LIN {X 0,Y 608.537,Z 464.117,A -85,B 0,C 180,E1 -528.614,E2 -528.614} C_VEL
LIN {X 0,Y 608.512,Z 476.576,A -85,B 0,C 180,E1 -529.025,E2 -529.025} C_VEL
LIN {X 0,Y 608.516,Z 487.728,A -85,B 0,C 180,E1 -529.519,E2 -529.519} C_VEL
LIN {X 0,Y 608.469,Z 499.507,A -85,B 0,C 180,E1 -530.191,E2 -530.191} C_VEL
LIN {X 0,Y 608.485,Z 510.019,A -85,B 0,C 180,E1 -530.946,E2 -530.946} C_VEL
LIN {X 0,Y 608.475,Z 518.633,A -85,B 0,C 180,E1 -531.699,E2 -531.699} C_VEL
LIN {X 0,Y 608.471,Z 526.564,A -85,B 0,C 180,E1 -532.534,E2 -532.534} C_VEL
LIN {X 0,Y 608.468,Z 534.069,A -85,B 0,C 180,E1 -533.497,E2 -533.497} C_VEL
LIN {X 0,Y 608.451,Z 539.606,A -85,B 0,C 180,E1 -534.366,E2 -534.366} C_VEL
LIN {X 0,Y 608.431,Z 544.75,A -85,B 0,C 180,E1 -535.362,E2 -535.362} C_VEL
LIN {X 0,Y 608.45,Z 548.74,A -85,B 0,C 180,E1 -536.358,E2 -536.358} C_VEL
LIN {X 0,Y 608.425,Z 551.691,A -85,B 0,C 180,E1 -537.352,E2 -537.352} C_VEL
LIN {X 0,Y 608.442,Z 553.127,A -85,B 0,C 180,E1 -538.014,E2 -538.014} C_VEL
LIN {X 0,Y 608.439,Z 554.752,A -85,B 0,C 180,E1 -539.338,E2 -539.338} C_VEL
LIN {X 0,Y 608.434,Z 554.995,A -85,B 0,C 180,E1 -540,E2 -540} C_VEL
LIN {X 0,Y 608.439,Z 554.815,A -85,B 0,C 180,E1 -540.662,E2 -540.662} C_VEL
LIN {X 0,Y 608.441,Z 553.277,A -85,B 0,C 180,E1 -541.986,E2 -541.986} C_VEL
LIN {X 0,Y 608.426,Z 551.918,A -85,B 0,C 180,E1 -542.648,E2 -542.648} C_VEL
LIN {X 0,Y 608.45,Z 549.042,A -85,B 0,C 180,E1 -543.642,E2 -543.642} C_VEL
LIN {X 0,Y 608.433,Z 545.144,A -85,B 0,C 180,E1 -544.638,E2 -544.638} C_VEL
LIN {X 0,Y 608.449,Z 540.113,A -85,B 0,C 180,E1 -545.634,E2 -545.634} C_VEL
LIN {X 0,Y 608.442,Z 533.793,A -85,B 0,C 180,E1 -546.633,E2 -546.633} C_VEL
LIN {X 0,Y 608.475,Z 525.88,A -85,B 0,C 180,E1 -547.633,E2 -547.633} C_VEL
LIN {X 0,Y 608.472,Z 516.032,A -85,B 0,C 180,E1 -548.636,E2 -548.636} C_VEL
LIN {X 0,Y 608.477,Z 513.929,A -85,B 0,C 180,E1 -548.82,E2 -548.82} C_VEL
LIN {X 0,Y 607.81,Z 509.588,A -85,B 0,C 180,E1 -549.19,E2 -549.19} C_VEL
LIN {X 0,Y 604.968,Z 502.332,A -85,B 0,C 180,E1 -549.77,E2 -549.77} C_VEL
LIN {X 0,Y 602.15,Z 494.692,A -85,B 0,C 180,E1 -550.302,E2 -550.302} C_VEL
LIN {X 0,Y 601.522,Z 489.64,A -85,B 0,C 180,E1 -550.595,E2 -550.595} C_VEL
LIN {X 0,Y 601.541,Z 478.352,A -85,B 0,C 180,E1 -551.124,E2 -551.124} C_VEL
LIN {X 0,Y 601.589,Z 465.836,A -85,B 0,C 180,E1 -551.562,E2 -551.562} C_VEL
LIN {X 0,Y 601.625,Z 452.229,A -85,B 0,C 180,E1 -551.882,E2 -551.882} C_VEL
LIN {X 0,Y 601.646,Z 413.087,A -85,B 0,C 180,E1 -552.373,E2 -552.373} C_VEL
LIN {X 0,Y 601.611,Z 346.67,A -85,B 0,C 180,E1 -553.17,E2 -553.17} C_VEL
LIN {X 0,Y 601.406,Z 345.276,A -85,B 0,C 180,E1 -553.215,E2 -553.215} C_VEL
LIN {X 0,Y 601.404,Z 331.568,A -85,B 0,C 180,E1 -555.939,E2 -555.939} C_VEL
LIN {X 0,Y 601.403,Z 331.566,A -85,B 0,C 180,E1 -558.392,E2 -558.392} C_VEL
LIN {X 0,Y 601.41,Z 331.574,A -85,B 0,C 180,E1 -561.239,E2 -561.239} C_VEL
LIN {X 0,Y 601.453,Z 331.56,A -85,B 0,C 180,E1 -564.141,E2 -564.141} C_VEL
LIN {X 0,Y 601.455,Z 331.568,A -85,B 0,C 180,E1 -567.111,E2 -567.111} C_VEL
LIN {X 0,Y 601.418,Z 331.571,A -85,B 0,C 180,E1 -569.393,E2 -569.393} C_VEL
LIN {X 0,Y 601.405,Z 331.568,A -85,B 0,C 180,E1 -571.727,E2 -571.727} C_VEL
LIN {X 0,Y 601.431,Z 331.562,A -85,B 0,C 180,E1 -574.118,E2 -574.118} C_VEL
LIN {X 0,Y 601.441,Z 331.567,A -85,B 0,C 180,E1 -577.382,E2 -577.382} C_VEL
LIN {X 0,Y 601.406,Z 331.565,A -85,B 0,C 180,E1 -579.996,E2 -579.996} C_VEL
LIN {X 0,Y 601.418,Z 331.568,A -85,B 0,C 180,E1 -582.67,E2 -582.67} C_VEL
LIN {X 0,Y 601.431,Z 331.566,A -85,B 0,C 180,E1 -585.482,E2 -585.482} C_VEL
LIN {X 0,Y 601.426,Z 331.565,A -85,B 0,C 180,E1 -588.407,E2 -588.407} C_VEL
LIN {X 0,Y 601.441,Z 331.57,A -85,B 0,C 180,E1 -590.875,E2 -590.875} C_VEL
LIN {X 0,Y 601.409,Z 331.568,A -85,B 0,C 180,E1 -593.417,E2 -593.417} C_VEL
LIN {X 0,Y 601.436,Z 331.562,A -85,B 0,C 180,E1 -596.064,E2 -596.064} C_VEL
LIN {X 0,Y 601.434,Z 331.569,A -85,B 0,C 180,E1 -599.058,E2 -599.058} C_VEL
LIN {X 0,Y 601.43,Z 331.565,A -85,B 0,C 180,E1 -601.372,E2 -601.372} C_VEL
LIN {X 0,Y 601.405,Z 331.566,A -85,B 0,C 180,E1 -603.636,E2 -603.636} C_VEL
LIN {X 0,Y 601.423,Z 331.57,A -85,B 0,C 180,E1 -606.589,E2 -606.589} C_VEL
LIN {X 0,Y 601.429,Z 331.563,A -85,B 0,C 180,E1 -609.477,E2 -609.477} C_VEL
LIN {X 0,Y 601.406,Z 331.569,A -85,B 0,C 180,E1 -612.311,E2 -612.311} C_VEL
LIN {X 0,Y 601.431,Z 331.566,A -85,B 0,C 180,E1 -615.102,E2 -615.102} C_VEL
LIN {X 0,Y 601.419,Z 331.564,A -85,B 0,C 180,E1 -617.857,E2 -617.857} C_VEL
LIN {X 0,Y 601.426,Z 331.573,A -85,B 0,C 180,E1 -620.584,E2 -620.584} C_VEL
LIN {X 0,Y 601.418,Z 331.564,A -85,B 0,C 180,E1 -623.357,E2 -623.357} C_VEL
LIN {X 0,Y 601.411,Z 331.566,A -85,B 0,C 180,E1 -625.979,E2 -625.979} C_VEL
LIN {X 0,Y 601.433,Z 331.571,A -85,B 0,C 180,E1 -628.66,E2 -628.66} C_VEL
LIN {X 0,Y 601.42,Z 331.564,A -85,B 0,C 180,E1 -631.338,E2 -631.338} C_VEL
LIN {X 0,Y 601.412,Z 331.568,A -85,B 0,C 180,E1 -634.02,E2 -634.02} C_VEL
LIN {X 0,Y 601.456,Z 331.565,A -85,B 0,C 180,E1 -636.709,E2 -636.709} C_VEL
LIN {X 0,Y 601.415,Z 331.564,A -85,B 0,C 180,E1 -639.415,E2 -639.415} C_VEL
LIN {X 0,Y 601.42,Z 331.57,A -85,B 0,C 180,E1 -642.142,E2 -642.142} C_VEL
LIN {X 0,Y 601.432,Z 331.564,A -85,B 0,C 180,E1 -644.896,E2 -644.896} C_VEL
LIN {X 0,Y 601.433,Z 331.563,A -85,B 0,C 180,E1 -646.985,E2 -646.985} C_VEL
LIN {X 0,Y 601.407,Z 331.568,A -85,B 0,C 180,E1 -649.808,E2 -649.808} C_VEL
LIN {X 0,Y 601.415,Z 331.569,A -85,B 0,C 180,E1 -652.605,E2 -652.605} C_VEL
LIN {X 0,Y 601.404,Z 331.567,A -85,B 0,C 180,E1 -654.877,E2 -654.877} C_VEL
LIN {X 0,Y 601.422,Z 331.568,A -85,B 0,C 180,E1 -657.866,E2 -657.866} C_VEL
LIN {X 0,Y 601.447,Z 331.57,A -85,B 0,C 180,E1 -660.162,E2 -660.162} C_VEL
LIN {X 0,Y 601.422,Z 331.565,A -85,B 0,C 180,E1 -662.715,E2 -662.715} C_VEL
LIN {X 0,Y 601.416,Z 331.564,A -85,B 0,C 180,E1 -665.115,E2 -665.115} C_VEL
LIN {X 0,Y 601.431,Z 331.563,A -85,B 0,C 180,E1 -667.418,E2 -667.418} C_VEL
LIN {X 0,Y 601.414,Z 331.573,A -85,B 0,C 180,E1 -669.993,E2 -669.993} C_VEL
LIN {X 0,Y 601.408,Z 331.567,A -85,B 0,C 180,E1 -672.669,E2 -672.669} C_VEL
LIN {X 0,Y 601.419,Z 331.566,A -85,B 0,C 180,E1 -675.481,E2 -675.481} C_VEL
LIN {X 0,Y 601.425,Z 331.567,A -85,B 0,C 180,E1 -678.405,E2 -678.405} C_VEL
LIN {X 0,Y 601.431,Z 331.562,A -85,B 0,C 180,E1 -680.875,E2 -680.875} C_VEL
LIN {X 0,Y 601.438,Z 331.568,A -85,B 0,C 180,E1 -683.733,E2 -683.733} C_VEL
LIN {X 0,Y 601.428,Z 331.563,A -85,B 0,C 180,E1 -686.687,E2 -686.687} C_VEL
LIN {X 0,Y 601.427,Z 331.563,A -85,B 0,C 180,E1 -689.058,E2 -689.058} C_VEL
LIN {X 0,Y 601.43,Z 331.565,A -85,B 0,C 180,E1 -691.373,E2 -691.373} C_VEL
LIN {X 0,Y 601.403,Z 331.573,A -85,B 0,C 180,E1 -693.636,E2 -693.636} C_VEL
LIN {X 0,Y 601.417,Z 331.564,A -85,B 0,C 180,E1 -696.59,E2 -696.59} C_VEL
LIN {X 0,Y 601.429,Z 331.568,A -85,B 0,C 180,E1 -699.478,E2 -699.478} C_VEL
LIN {X 0,Y 601.397,Z 331.568,A -85,B 0,C 180,E1 -702.312,E2 -702.312} C_VEL
LIN {X 0,Y 601.412,Z 331.565,A -85,B 0,C 180,E1 -704.409,E2 -704.409} C_VEL
LIN {X 0,Y 601.419,Z 331.566,A -85,B 0,C 180,E1 -707.172,E2 -707.172} C_VEL
LIN {X 0,Y 601.431,Z 331.568,A -85,B 0,C 180,E1 -709.905,E2 -709.905} C_VEL
LIN {X 0,Y 601.446,Z 331.56,A -85,B 0,C 180,E1 -712.615,E2 -712.615} C_VEL
LIN {X 0,Y 601.426,Z 331.569,A -85,B 0,C 180,E1 -715.308,E2 -715.308} C_VEL
LIN {X 0,Y 601.418,Z 331.567,A -85,B 0,C 180,E1 -717.991,E2 -717.991} C_VEL
LIN {X 0,Y 601.449,Z 331.56,A -85,B 0,C 180,E1 -720.67,E2 -720.67} C_VEL
LIN {X 0,Y 601.428,Z 331.571,A -85,B 0,C 180,E1 -723.35,E2 -723.35} C_VEL
LIN {X 0,Y 601.404,Z 331.567,A -85,B 0,C 180,E1 -726.037,E2 -726.037} C_VEL
LIN {X 0,Y 601.434,Z 331.563,A -85,B 0,C 180,E1 -728.738,E2 -728.738} C_VEL
LIN {X 0,Y 601.428,Z 331.572,A -85,B 0,C 180,E1 -731.458,E2 -731.458} C_VEL
LIN {X 0,Y 601.411,Z 331.565,A -85,B 0,C 180,E1 -734.206,E2 -734.206} C_VEL
LIN {X 0,Y 601.43,Z 331.567,A -85,B 0,C 180,E1 -736.986,E2 -736.986} C_VEL
LIN {X 0,Y 601.404,Z 331.568,A -85,B 0,C 180,E1 -739.81,E2 -739.81} C_VEL
LIN {X 0,Y 601.406,Z 331.567,A -85,B 0,C 180,E1 -742.683,E2 -742.683} C_VEL
LIN {X 0,Y 601.401,Z 331.57,A -85,B 0,C 180,E1 -744.879,E2 -744.879} C_VEL
LIN {X 0,Y 601.419,Z 331.565,A -85,B 0,C 180,E1 -747.868,E2 -747.868} C_VEL
LIN {X 0,Y 601.42,Z 331.563,A -85,B 0,C 180,E1 -750.165,E2 -750.165} C_VEL
LIN {X 0,Y 601.425,Z 331.566,A -85,B 0,C 180,E1 -752.718,E2 -752.718} C_VEL
LIN {X 0,Y 601.408,Z 331.576,A -85,B 0,C 180,E1 -755.116,E2 -755.116} C_VEL
LIN {X 0,Y 601.432,Z 331.567,A -85,B 0,C 180,E1 -757.419,E2 -757.419} C_VEL
LIN {X 0,Y 601.409,Z 331.565,A -85,B 0,C 180,E1 -759.995,E2 -759.995} C_VEL
LIN {X 0,Y 601.435,Z 331.566,A -85,B 0,C 180,E1 -762.668,E2 -762.668} C_VEL
LIN {X 0,Y 601.42,Z 331.566,A -85,B 0,C 180,E1 -765.483,E2 -765.483} C_VEL
LIN {X 0,Y 601.423,Z 331.565,A -85,B 0,C 180,E1 -768.407,E2 -768.407} C_VEL
LIN {X 0,Y 601.439,Z 331.57,A -85,B 0,C 180,E1 -770.877,E2 -770.877} C_VEL
LIN {X 0,Y 601.442,Z 331.561,A -85,B 0,C 180,E1 -773.735,E2 -773.735} C_VEL
LIN {X 0,Y 601.432,Z 331.562,A -85,B 0,C 180,E1 -776.065,E2 -776.065} C_VEL
LIN {X 0,Y 601.431,Z 331.569,A -85,B 0,C 180,E1 -779.06,E2 -779.06} C_VEL
LIN {X 0,Y 601.429,Z 331.565,A -85,B 0,C 180,E1 -781.374,E2 -781.374} C_VEL
LIN {X 0,Y 601.404,Z 331.567,A -85,B 0,C 180,E1 -783.637,E2 -783.637} C_VEL
LIN {X 0,Y 601.44,Z 331.583,A -85,B 0,C 180,E1 -785.658,E2 -785.658} C_VEL
LIN {X 0,Y 601.762,Z 334.596,A -85,B 0,C 180,E1 -786.057,E2 -786.057} C_VEL
LIN {X 0,Y 601.686,Z 356.122,A -85,B 0,C 180,E1 -788.772,E2 -788.772} C_VEL
LIN {X 0,Y 601.603,Z 379.082,A -85,B 0,C 180,E1 -791.615,E2 -791.615} C_VEL
LIN {X 0,Y 601.529,Z 403.477,A -85,B 0,C 180,E1 -794.586,E2 -794.586} C_VEL
LIN {X 0,Y 601.469,Z 421.953,A -85,B 0,C 180,E1 -796.809,E2 -796.809} C_VEL
LIN {X 0,Y 601.657,Z 435.738,A -85,B 0,C 180,E1 -796.985,E2 -796.985} C_VEL
LIN {X 0,Y 601.604,Z 530.994,A -85,B 0,C 180,E1 -798.14,E2 -798.14} C_VEL
LIN {X 0,Y 601.573,Z 544.248,A -85,B 0,C 180,E1 -798.439,E2 -798.439} C_VEL
LIN {X 0,Y 601.543,Z 555.978,A -85,B 0,C 180,E1 -798.828,E2 -798.828} C_VEL
LIN {X 0,Y 601.515,Z 566.941,A -85,B 0,C 180,E1 -799.312,E2 -799.312} C_VEL
LIN {X 0,Y 601.479,Z 577.595,A -85,B 0,C 180,E1 -799.907,E2 -799.907} C_VEL
LIN {X 0,Y 601.446,Z 588.486,A -85,B 0,C 180,E1 -800.67,E2 -800.67} C_VEL
LIN {X 0,Y 601.429,Z 599.121,A -85,B 0,C 180,E1 -801.602,E2 -801.602} C_VEL
LIN {X 0,Y 601.417,Z 606.968,A -85,B 0,C 180,E1 -802.447,E2 -802.447} C_VEL
LIN {X 0,Y 601.369,Z 614.229,A -85,B 0,C 180,E1 -803.399,E2 -803.399} C_VEL
LIN {X 0,Y 601.371,Z 619.871,A -85,B 0,C 180,E1 -804.3,E2 -804.3} C_VEL
LIN {X 0,Y 601.337,Z 624.953,A -85,B 0,C 180,E1 -805.308,E2 -805.308} C_VEL
LIN {X 0,Y 601.367,Z 628.899,A -85,B 0,C 180,E1 -806.315,E2 -806.315} C_VEL
LIN {X 0,Y 601.325,Z 631.811,A -85,B 0,C 180,E1 -807.321,E2 -807.321} C_VEL
LIN {X 0,Y 601.341,Z 633.203,A -85,B 0,C 180,E1 -807.991,E2 -807.991} C_VEL
LIN {X 0,Y 601.339,Z 634.784,A -85,B 0,C 180,E1 -809.331,E2 -809.331} C_VEL
LIN {X 0,Y 601.335,Z 635,A -85,B 0,C 180,E1 -810.001,E2 -810.001} C_VEL
LIN {X 0,Y 601.348,Z 634.183,A -85,B 0,C 180,E1 -811.34,E2 -811.34} C_VEL
LIN {X 0,Y 601.342,Z 633.201,A -85,B 0,C 180,E1 -812.01,E2 -812.01} C_VEL
LIN {X 0,Y 601.325,Z 631.807,A -85,B 0,C 180,E1 -812.68,E2 -812.68} C_VEL
LIN {X 0,Y 601.367,Z 628.894,A -85,B 0,C 180,E1 -813.686,E2 -813.686} C_VEL
LIN {X 0,Y 601.337,Z 624.947,A -85,B 0,C 180,E1 -814.693,E2 -814.693} C_VEL
LIN {X 0,Y 601.372,Z 618.873,A -85,B 0,C 180,E1 -815.87,E2 -815.87} C_VEL
LIN {X 0,Y 601.382,Z 612.23,A -85,B 0,C 180,E1 -816.88,E2 -816.88} C_VEL
LIN {X 0,Y 601.401,Z 603.983,A -85,B 0,C 180,E1 -817.893,E2 -817.893} C_VEL
LIN {X 0,Y 601.436,Z 595.529,A -85,B 0,C 180,E1 -818.738,E2 -818.738} C_VEL
LIN {X 0,Y 601.442,Z 585.083,A -85,B 0,C 180,E1 -819.586,E2 -819.586} C_VEL
LIN {X 0,Y 601.472,Z 574.746,A -85,B 0,C 180,E1 -820.265,E2 -820.265} C_VEL
LIN {X 0,Y 601.536,Z 563.894,A -85,B 0,C 180,E1 -820.836,E2 -820.836} C_VEL
LIN {X 0,Y 601.557,Z 551.36,A -85,B 0,C 180,E1 -821.341,E2 -821.341} C_VEL
LIN {X 0,Y 601.569,Z 538.322,A -85,B 0,C 180,E1 -821.712,E2 -821.712} C_VEL
LIN {X 0,Y 601.614,Z 525.03,A -85,B 0,C 180,E1 -821.947,E2 -821.947} C_VEL
LIN {X 0,Y 601.617,Z 423.085,A -85,B 0,C 180,E1 -823.168,E2 -823.168} C_VEL
LIN {X 0,Y 601.462,Z 421.76,A -85,B 0,C 180,E1 -823.214,E2 -823.214} C_VEL
LIN {X 0,Y 601.546,Z 399.159,A -85,B 0,C 180,E1 -825.936,E2 -825.936} C_VEL
LIN {X 0,Y 601.634,Z 375.064,A -85,B 0,C 180,E1 -828.878,E2 -828.878} C_VEL
LIN {X 0,Y 601.696,Z 351.803,A -85,B 0,C 180,E1 -831.769,E2 -831.769} C_VEL
LIN {X 0,Y 601.751,Z 333.148,A -85,B 0,C 180,E1 -834.128,E2 -834.128} C_VEL
LIN {X 0,Y 601.422,Z 331.568,A -85,B 0,C 180,E1 -834.362,E2 -834.362} C_VEL
LIN {X 0,Y 601.458,Z 331.569,A -85,B 0,C 180,E1 -837.111,E2 -837.111} C_VEL
LIN {X 0,Y 601.427,Z 331.569,A -85,B 0,C 180,E1 -839.393,E2 -839.393} C_VEL
LIN {X 0,Y 601.416,Z 331.566,A -85,B 0,C 180,E1 -841.727,E2 -841.727} C_VEL
LIN {X 0,Y 601.434,Z 331.562,A -85,B 0,C 180,E1 -844.119,E2 -844.119} C_VEL
LIN {X 0,Y 601.409,Z 331.568,A -85,B 0,C 180,E1 -846.583,E2 -846.583} C_VEL
LIN {X 0,Y 601.447,Z 331.563,A -85,B 0,C 180,E1 -849.536,E2 -849.536} C_VEL
LIN {X 0,Y 601.412,Z 331.568,A -85,B 0,C 180,E1 -852.59,E2 -852.59} C_VEL
LIN {X 0,Y 601.432,Z 331.565,A -85,B 0,C 180,E1 -855.482,E2 -855.482} C_VEL
LIN {X 0,Y 601.428,Z 331.564,A -85,B 0,C 180,E1 -858.407,E2 -858.407} C_VEL
LIN {X 0,Y 601.435,Z 331.563,A -85,B 0,C 180,E1 -861.529,E2 -861.529} C_VEL
LIN {X 0,Y 601.389,Z 331.568,A -85,B 0,C 180,E1 -864.245,E2 -864.245} C_VEL
LIN {X 0,Y 601.423,Z 331.57,A -85,B 0,C 180,E1 -866.686,E2 -866.686} C_VEL
LIN {X 0,Y 601.418,Z 331.571,A -85,B 0,C 180,E1 -869.058,E2 -869.058} C_VEL
LIN {X 0,Y 601.436,Z 331.564,A -85,B 0,C 180,E1 -871.373,E2 -871.373} C_VEL
LIN {X 0,Y 601.407,Z 331.566,A -85,B 0,C 180,E1 -873.636,E2 -873.636} C_VEL
LIN {X 0,Y 601.419,Z 331.571,A -85,B 0,C 180,E1 -876.589,E2 -876.589} C_VEL
LIN {X 0,Y 601.433,Z 331.563,A -85,B 0,C 180,E1 -879.478,E2 -879.478} C_VEL
LIN {X 0,Y 601.399,Z 331.57,A -85,B 0,C 180,E1 -882.312,E2 -882.312} C_VEL
LIN {X 0,Y 601.427,Z 331.729,A -85,B 0,C 180,E1 -884.192,E2 -884.192} C_VEL
LIN {X 0,Y 601.403,Z 345.363,A -85,B 0,C 180,E1 -886.892,E2 -886.892} C_VEL
LIN {X 0,Y 601.677,Z 350.116,A -85,B 0,C 180,E1 -886.963,E2 -886.963} C_VEL
LIN {X 0,Y 601.627,Z 450.826,A -85,B 0,C 180,E1 -888.182,E2 -888.182} C_VEL
LIN {X 0,Y 601.601,Z 464.145,A -85,B 0,C 180,E1 -888.481,E2 -888.481} C_VEL
LIN {X 0,Y 601.54,Z 476.533,A -85,B 0,C 180,E1 -888.895,E2 -888.895} C_VEL
LIN {X 0,Y 601.541,Z 487.735,A -85,B 0,C 180,E1 -889.396,E2 -889.396} C_VEL
LIN {X 0,Y 601.47,Z 499.512,A -85,B 0,C 180,E1 -890.075,E2 -890.075} C_VEL
LIN {X 0,Y 601.444,Z 510.021,A -85,B 0,C 180,E1 -890.839,E2 -890.839} C_VEL
LIN {X 0,Y 601.429,Z 518.638,A -85,B 0,C 180,E1 -891.601,E2 -891.601} C_VEL
LIN {X 0,Y 601.418,Z 526.571,A -85,B 0,C 180,E1 -892.446,E2 -892.446} C_VEL
LIN {X 0,Y 601.377,Z 533.879,A -85,B 0,C 180,E1 -893.393,E2 -893.393} C_VEL
LIN {X 0,Y 601.372,Z 539.601,A -85,B 0,C 180,E1 -894.299,E2 -894.299} C_VEL
LIN {X 0,Y 601.335,Z 544.748,A -85,B 0,C 180,E1 -895.307,E2 -895.307} C_VEL
LIN {X 0,Y 601.368,Z 548.741,A -85,B 0,C 180,E1 -896.315,E2 -896.315} C_VEL
LIN {X 0,Y 601.324,Z 551.693,A -85,B 0,C 180,E1 -897.32,E2 -897.32} C_VEL
LIN {X 0,Y 601.341,Z 553.13,A -85,B 0,C 180,E1 -897.991,E2 -897.991} C_VEL
LIN {X 0,Y 601.339,Z 554.754,A -85,B 0,C 180,E1 -899.33,E2 -899.33} C_VEL
LIN {X 0,Y 601.335,Z 554.996,A -85,B 0,C 180,E1 -900,E2 -900} C_VEL
LIN {X 0,Y 601.339,Z 554.817,A -85,B 0,C 180,E1 -900.67,E2 -900.67} C_VEL
LIN {X 0,Y 601.34,Z 553.278,A -85,B 0,C 180,E1 -902.009,E2 -902.009} C_VEL
LIN {X 0,Y 601.326,Z 551.916,A -85,B 0,C 180,E1 -902.679,E2 -902.679} C_VEL
LIN {X 0,Y 601.368,Z 549.042,A -85,B 0,C 180,E1 -903.685,E2 -903.685} C_VEL
LIN {X 0,Y 601.337,Z 545.144,A -85,B 0,C 180,E1 -904.693,E2 -904.693} C_VEL
LIN {X 0,Y 601.373,Z 540.111,A -85,B 0,C 180,E1 -905.701,E2 -905.701} C_VEL
LIN {X 0,Y 601.383,Z 533.782,A -85,B 0,C 180,E1 -906.711,E2 -906.711} C_VEL
LIN {X 0,Y 601.396,Z 525.878,A -85,B 0,C 180,E1 -907.723,E2 -907.723} C_VEL
LIN {X 0,Y 601.422,Z 517.808,A -85,B 0,C 180,E1 -908.568,E2 -908.568} C_VEL
LIN {X 0,Y 601.452,Z 507.963,A -85,B 0,C 180,E1 -909.415,E2 -909.415} C_VEL
LIN {X 0,Y 601.481,Z 496.919,A -85,B 0,C 180,E1 -910.179,E2 -910.179} C_VEL
LIN {X 0,Y 601.522,Z 489.64,A -85,B 0,C 180,E1 -910.595,E2 -910.595} C_VEL
LIN {X 0,Y 600.883,Z 484.509,A -85,B 0,C 180,E1 -910.869,E2 -910.869} C_VEL
LIN {X 0,Y 598.037,Z 476.063,A -85,B 0,C 180,E1 -911.29,E2 -911.29} C_VEL
LIN {X 0,Y 595.225,Z 467.317,A -85,B 0,C 180,E1 -911.644,E2 -911.644} C_VEL
LIN {X 0,Y 594.631,Z 461.725,A -85,B 0,C 180,E1 -911.813,E2 -911.813} C_VEL
LIN {X 0,Y 594.697,Z 448.231,A -85,B 0,C 180,E1 -912.087,E2 -912.087} C_VEL
LIN {X 0,Y 594.715,Z 347.518,A -85,B 0,C 180,E1 -913.315,E2 -913.315} C_VEL
LIN {X 0,Y 594.382,Z 345.273,A -85,B 0,C 180,E1 -913.374,E2 -913.374} C_VEL
LIN {X 0,Y 594.388,Z 332.443,A -85,B 0,C 180,E1 -915.956,E2 -915.956} C_VEL
LIN {X 0,Y 594.379,Z 332.442,A -85,B 0,C 180,E1 -918.618,E2 -918.618} C_VEL
LIN {X 0,Y 594.37,Z 332.449,A -85,B 0,C 180,E1 -921.503,E2 -921.503} C_VEL
LIN {X 0,Y 594.393,Z 332.439,A -85,B 0,C 180,E1 -924.446,E2 -924.446} C_VEL
LIN {X 0,Y 594.388,Z 332.442,A -85,B 0,C 180,E1 -926.699,E2 -926.699} C_VEL
LIN {X 0,Y 594.385,Z 332.447,A -85,B 0,C 180,E1 -928.998,E2 -928.998} C_VEL
LIN {X 0,Y 594.381,Z 332.444,A -85,B 0,C 180,E1 -931.642,E2 -931.642} C_VEL
LIN {X 0,Y 594.382,Z 332.442,A -85,B 0,C 180,E1 -934.58,E2 -934.58} C_VEL
LIN {X 0,Y 594.394,Z 332.442,A -85,B 0,C 180,E1 -937.608,E2 -937.608} C_VEL
LIN {X 0,Y 594.372,Z 332.444,A -85,B 0,C 180,E1 -940.567,E2 -940.567} C_VEL
LIN {X 0,Y 594.372,Z 332.448,A -85,B 0,C 180,E1 -943.299,E2 -943.299} C_VEL
LIN {X 0,Y 594.372,Z 332.442,A -85,B 0,C 180,E1 -946.16,E2 -946.16} C_VEL
LIN {X 0,Y 594.38,Z 332.448,A -85,B 0,C 180,E1 -949.178,E2 -949.178} C_VEL
LIN {X 0,Y 594.389,Z 332.44,A -85,B 0,C 180,E1 -952.059,E2 -952.059} C_VEL
LIN {X 0,Y 594.366,Z 332.448,A -85,B 0,C 180,E1 -954.675,E2 -954.675} C_VEL
LIN {X 0,Y 594.38,Z 332.448,A -85,B 0,C 180,E1 -957.088,E2 -957.088} C_VEL
LIN {X 0,Y 594.392,Z 332.44,A -85,B 0,C 180,E1 -959.671,E2 -959.671} C_VEL
LIN {X 0,Y 594.379,Z 332.446,A -85,B 0,C 180,E1 -962.539,E2 -962.539} C_VEL
LIN {X 0,Y 594.381,Z 332.451,A -85,B 0,C 180,E1 -964.807,E2 -964.807} C_VEL
LIN {X 0,Y 594.369,Z 332.445,A -85,B 0,C 180,E1 -967.264,E2 -967.264} C_VEL
LIN {X 0,Y 594.376,Z 332.441,A -85,B 0,C 180,E1 -969.946,E2 -969.946} C_VEL
LIN {X 0,Y 594.39,Z 332.449,A -85,B 0,C 180,E1 -972.806,E2 -972.806} C_VEL
LIN {X 0,Y 594.394,Z 332.439,A -85,B 0,C 180,E1 -975.825,E2 -975.825} C_VEL
LIN {X 0,Y 594.399,Z 332.444,A -85,B 0,C 180,E1 -978.404,E2 -978.404} C_VEL
LIN {X 0,Y 594.383,Z 332.443,A -85,B 0,C 180,E1 -981.157,E2 -981.157} C_VEL
LIN {X 0,Y 594.387,Z 332.441,A -85,B 0,C 180,E1 -983.891,E2 -983.891} C_VEL
LIN {X 0,Y 594.39,Z 332.449,A -85,B 0,C 180,E1 -986.61,E2 -986.61} C_VEL
LIN {X 0,Y 594.419,Z 332.436,A -85,B 0,C 180,E1 -989.322,E2 -989.322} C_VEL
LIN {X 0,Y 594.406,Z 332.44,A -85,B 0,C 180,E1 -992.032,E2 -992.032} C_VEL
LIN {X 0,Y 594.399,Z 332.444,A -85,B 0,C 180,E1 -994.747,E2 -994.747} C_VEL
LIN {X 0,Y 594.395,Z 332.439,A -85,B 0,C 180,E1 -997.472,E2 -997.472} C_VEL
LIN {X 0,Y 594.399,Z 332.445,A -85,B 0,C 180,E1 -1000.215,E2 -1000.215} C_VEL
LIN {X 0,Y 594.367,Z 332.444,A -85,B 0,C 180,E1 -1002.982,E2 -1002.982} C_VEL
LIN {X 0,Y 594.369,Z 332.444,A -85,B 0,C 180,E1 -1005.78,E2 -1005.78} C_VEL
LIN {X 0,Y 594.388,Z 332.445,A -85,B 0,C 180,E1 -1008.616,E2 -1008.616} C_VEL
LIN {X 0,Y 594.367,Z 332.443,A -85,B 0,C 180,E1 -1011.502,E2 -1011.502} C_VEL
LIN {X 0,Y 594.388,Z 332.447,A -85,B 0,C 180,E1 -1014.445,E2 -1014.445} C_VEL
LIN {X 0,Y 594.385,Z 332.443,A -85,B 0,C 180,E1 -1016.698,E2 -1016.698} C_VEL
LIN {X 0,Y 594.382,Z 332.441,A -85,B 0,C 180,E1 -1018.997,E2 -1018.997} C_VEL
LIN {X 0,Y 594.391,Z 332.442,A -85,B 0,C 180,E1 -1021.645,E2 -1021.645} C_VEL
LIN {X 0,Y 594.398,Z 332.442,A -85,B 0,C 180,E1 -1024.578,E2 -1024.578} C_VEL
LIN {X 0,Y 594.383,Z 332.44,A -85,B 0,C 180,E1 -1027.086,E2 -1027.086} C_VEL
LIN {X 0,Y 594.377,Z 332.446,A -85,B 0,C 180,E1 -1029.774,E2 -1029.774} C_VEL
LIN {X 0,Y 594.367,Z 332.447,A -85,B 0,C 180,E1 -1032.374,E2 -1032.374} C_VEL
LIN {X 0,Y 594.356,Z 332.444,A -85,B 0,C 180,E1 -1035.19,E2 -1035.19} C_VEL
LIN {X 0,Y 594.384,Z 332.444,A -85,B 0,C 180,E1 -1037.626,E2 -1037.626} C_VEL
LIN {X 0,Y 594.388,Z 332.444,A -85,B 0,C 180,E1 -1040.321,E2 -1040.321} C_VEL
LIN {X 0,Y 594.381,Z 332.44,A -85,B 0,C 180,E1 -1042.913,E2 -1042.913} C_VEL
LIN {X 0,Y 594.381,Z 332.45,A -85,B 0,C 180,E1 -1045.86,E2 -1045.86} C_VEL
LIN {X 0,Y 594.385,Z 332.44,A -85,B 0,C 180,E1 -1048.651,E2 -1048.651} C_VEL
LIN {X 0,Y 594.379,Z 332.441,A -85,B 0,C 180,E1 -1051.041,E2 -1051.041} C_VEL
LIN {X 0,Y 594.386,Z 332.448,A -85,B 0,C 180,E1 -1053.975,E2 -1053.975} C_VEL
LIN {X 0,Y 594.389,Z 332.442,A -85,B 0,C 180,E1 -1056.296,E2 -1056.296} C_VEL
LIN {X 0,Y 594.4,Z 332.44,A -85,B 0,C 180,E1 -1059.224,E2 -1059.224} C_VEL
LIN {X 0,Y 594.376,Z 332.445,A -85,B 0,C 180,E1 -1062.096,E2 -1062.096} C_VEL
LIN {X 0,Y 594.366,Z 332.445,A -85,B 0,C 180,E1 -1064.219,E2 -1064.219} C_VEL
LIN {X 0,Y 594.366,Z 332.443,A -85,B 0,C 180,E1 -1067.017,E2 -1067.017} C_VEL
LIN {X 0,Y 594.39,Z 332.447,A -85,B 0,C 180,E1 -1069.784,E2 -1069.784} C_VEL
LIN {X 0,Y 594.395,Z 332.439,A -85,B 0,C 180,E1 -1072.527,E2 -1072.527} C_VEL
LIN {X 0,Y 594.394,Z 332.444,A -85,B 0,C 180,E1 -1075.252,E2 -1075.252} C_VEL
LIN {X 0,Y 594.388,Z 332.443,A -85,B 0,C 180,E1 -1077.967,E2 -1077.967} C_VEL
LIN {X 0,Y 594.419,Z 332.436,A -85,B 0,C 180,E1 -1080.678,E2 -1080.678} C_VEL
LIN {X 0,Y 594.379,Z 332.449,A -85,B 0,C 180,E1 -1083.389,E2 -1083.389} C_VEL
LIN {X 0,Y 594.36,Z 332.444,A -85,B 0,C 180,E1 -1086.109,E2 -1086.109} C_VEL
LIN {X 0,Y 594.394,Z 332.44,A -85,B 0,C 180,E1 -1088.842,E2 -1088.842} C_VEL
LIN {X 0,Y 594.387,Z 332.447,A -85,B 0,C 180,E1 -1091.596,E2 -1091.596} C_VEL
LIN {X 0,Y 594.382,Z 332.44,A -85,B 0,C 180,E1 -1094.377,E2 -1094.377} C_VEL
LIN {X 0,Y 594.387,Z 332.448,A -85,B 0,C 180,E1 -1097.194,E2 -1097.194} C_VEL
LIN {X 0,Y 594.373,Z 332.442,A -85,B 0,C 180,E1 -1100.054,E2 -1100.054} C_VEL
LIN {X 0,Y 594.358,Z 332.449,A -85,B 0,C 180,E1 -1102.968,E2 -1102.968} C_VEL
LIN {X 0,Y 594.373,Z 332.451,A -85,B 0,C 180,E1 -1105.193,E2 -1105.193} C_VEL
LIN {X 0,Y 594.377,Z 332.446,A -85,B 0,C 180,E1 -1107.527,E2 -1107.527} C_VEL
LIN {X 0,Y 594.38,Z 332.441,A -85,B 0,C 180,E1 -1110.329,E2 -1110.329} C_VEL
LIN {X 0,Y 594.374,Z 332.448,A -85,B 0,C 180,E1 -1112.951,E2 -1112.951} C_VEL
LIN {X 0,Y 594.376,Z 332.447,A -85,B 0,C 180,E1 -1115.407,E2 -1115.407} C_VEL
LIN {X 0,Y 594.384,Z 332.44,A -85,B 0,C 180,E1 -1117.941,E2 -1117.941} C_VEL
LIN {X 0,Y 594.388,Z 332.446,A -85,B 0,C 180,E1 -1120.825,E2 -1120.825} C_VEL
LIN {X 0,Y 594.382,Z 332.446,A -85,B 0,C 180,E1 -1123.298,E2 -1123.298} C_VEL
LIN {X 0,Y 594.377,Z 332.441,A -85,B 0,C 180,E1 -1126.16,E2 -1126.16} C_VEL
LIN {X 0,Y 594.378,Z 332.448,A -85,B 0,C 180,E1 -1129.178,E2 -1129.178} C_VEL
LIN {X 0,Y 594.385,Z 332.44,A -85,B 0,C 180,E1 -1132.061,E2 -1132.061} C_VEL
LIN {X 0,Y 594.386,Z 332.446,A -85,B 0,C 180,E1 -1134.672,E2 -1134.672} C_VEL
LIN {X 0,Y 594.376,Z 332.448,A -85,B 0,C 180,E1 -1137.089,E2 -1137.089} C_VEL
LIN {X 0,Y 594.4,Z 332.439,A -85,B 0,C 180,E1 -1139.67,E2 -1139.67} C_VEL
LIN {X 0,Y 594.373,Z 332.448,A -85,B 0,C 180,E1 -1142.54,E2 -1142.54} C_VEL
LIN {X 0,Y 594.36,Z 332.451,A -85,B 0,C 180,E1 -1145.181,E2 -1145.181} C_VEL
LIN {X 0,Y 594.381,Z 332.517,A -85,B 0,C 180,E1 -1145.471,E2 -1145.471} C_VEL
LIN {X 0,Y 594.902,Z 336.031,A -85,B 0,C 180,E1 -1145.949,E2 -1145.949} C_VEL
LIN {X 0,Y 594.777,Z 357.408,A -85,B 0,C 180,E1 -1148.676,E2 -1148.676} C_VEL
LIN {X 0,Y 594.652,Z 379.082,A -85,B 0,C 180,E1 -1151.392,E2 -1151.392} C_VEL
LIN {X 0,Y 594.553,Z 403.477,A -85,B 0,C 180,E1 -1154.401,E2 -1154.401} C_VEL
LIN {X 0,Y 594.459,Z 421.953,A -85,B 0,C 180,E1 -1156.65,E2 -1156.65} C_VEL
LIN {X 0,Y 594.795,Z 426.794,A -85,B 0,C 180,E1 -1156.723,E2 -1156.723} C_VEL
LIN {X 0,Y 594.684,Z 530.994,A -85,B 0,C 180,E1 -1158,E2 -1158} C_VEL
LIN {X 0,Y 594.616,Z 544.249,A -85,B 0,C 180,E1 -1158.302,E2 -1158.302} C_VEL
LIN {X 0,Y 594.575,Z 557.21,A -85,B 0,C 180,E1 -1158.743,E2 -1158.743} C_VEL
LIN {X 0,Y 594.537,Z 568.649,A -85,B 0,C 180,E1 -1159.271,E2 -1159.271} C_VEL
LIN {X 0,Y 594.469,Z 580.213,A -85,B 0,C 180,E1 -1159.958,E2 -1159.958} C_VEL
LIN {X 0,Y 594.413,Z 590.607,A -85,B 0,C 180,E1 -1160.73,E2 -1160.73} C_VEL
LIN {X 0,Y 594.383,Z 599.121,A -85,B 0,C 180,E1 -1161.501,E2 -1161.501} C_VEL
LIN {X 0,Y 594.346,Z 606.968,A -85,B 0,C 180,E1 -1162.356,E2 -1162.356} C_VEL
LIN {X 0,Y 594.282,Z 614.817,A -85,B 0,C 180,E1 -1163.409,E2 -1163.409} C_VEL
LIN {X 0,Y 594.289,Z 621.685,A -85,B 0,C 180,E1 -1164.572,E2 -1164.572} C_VEL
LIN {X 0,Y 594.27,Z 626.375,A -85,B 0,C 180,E1 -1165.592,E2 -1165.592} C_VEL
LIN {X 0,Y 594.267,Z 629.959,A -85,B 0,C 180,E1 -1166.611,E2 -1166.611} C_VEL
LIN {X 0,Y 594.226,Z 631.811,A -85,B 0,C 180,E1 -1167.289,E2 -1167.289} C_VEL
LIN {X 0,Y 594.24,Z 633.203,A -85,B 0,C 180,E1 -1167.967,E2 -1167.967} C_VEL
LIN {X 0,Y 594.239,Z 634.785,A -85,B 0,C 180,E1 -1169.323,E2 -1169.323} C_VEL
LIN {X 0,Y 594.236,Z 635,A -85,B 0,C 180,E1 -1170.001,E2 -1170.001} C_VEL
LIN {X 0,Y 594.248,Z 634.184,A -85,B 0,C 180,E1 -1171.356,E2 -1171.356} C_VEL
LIN {X 0,Y 594.24,Z 633.2,A -85,B 0,C 180,E1 -1172.034,E2 -1172.034} C_VEL
LIN {X 0,Y 594.226,Z 631.808,A -85,B 0,C 180,E1 -1172.712,E2 -1172.712} C_VEL
LIN {X 0,Y 594.289,Z 628.894,A -85,B 0,C 180,E1 -1173.73,E2 -1173.73} C_VEL
LIN {X 0,Y 594.242,Z 624.946,A -85,B 0,C 180,E1 -1174.75,E2 -1174.75} C_VEL
LIN {X 0,Y 594.304,Z 618.873,A -85,B 0,C 180,E1 -1175.94,E2 -1175.94} C_VEL
LIN {X 0,Y 594.309,Z 612.231,A -85,B 0,C 180,E1 -1176.963,E2 -1176.963} C_VEL
LIN {X 0,Y 594.359,Z 603.983,A -85,B 0,C 180,E1 -1177.987,E2 -1177.987} C_VEL
LIN {X 0,Y 594.382,Z 595.529,A -85,B 0,C 180,E1 -1178.843,E2 -1178.843} C_VEL
LIN {X 0,Y 594.428,Z 585.084,A -85,B 0,C 180,E1 -1179.7,E2 -1179.7} C_VEL
LIN {X 0,Y 594.483,Z 574.747,A -85,B 0,C 180,E1 -1180.387,E2 -1180.387} C_VEL
LIN {X 0,Y 594.559,Z 563.706,A -85,B 0,C 180,E1 -1180.974,E2 -1180.974} C_VEL
LIN {X 0,Y 594.583,Z 551.689,A -85,B 0,C 180,E1 -1181.465,E2 -1181.465} C_VEL
LIN {X 0,Y 594.637,Z 538.321,A -85,B 0,C 180,E1 -1181.851,E2 -1181.851} C_VEL
LIN {X 0,Y 594.691,Z 525.03,A -85,B 0,C 180,E1 -1182.088,E2 -1182.088} C_VEL
LIN {X 0,Y 594.607,Z 423.085,A -85,B 0,C 180,E1 -1183.326,E2 -1183.326} C_VEL
LIN {X 0,Y 594.471,Z 421.76,A -85,B 0,C 180,E1 -1183.373,E2 -1183.373} C_VEL
LIN {X 0,Y 594.568,Z 399.159,A -85,B 0,C 180,E1 -1186.128,E2 -1186.128} C_VEL
LIN {X 0,Y 594.68,Z 375.057,A -85,B 0,C 180,E1 -1189.109,E2 -1189.109} C_VEL
LIN {X 0,Y 594.829,Z 351.803,A -85,B 0,C 180,E1 -1192.033,E2 -1192.033} C_VEL
LIN {X 0,Y 594.853,Z 334.583,A -85,B 0,C 180,E1 -1194.241,E2 -1194.241} C_VEL
LIN {X 0,Y 594.373,Z 332.448,A -85,B 0,C 180,E1 -1194.573,E2 -1194.573} C_VEL
LIN {X 0,Y 594.39,Z 332.443,A -85,B 0,C 180,E1 -1196.7,E2 -1196.7} C_VEL
LIN {X 0,Y 594.386,Z 332.448,A -85,B 0,C 180,E1 -1198.999,E2 -1198.999} C_VEL
LIN {X 0,Y 594.396,Z 332.442,A -85,B 0,C 180,E1 -1201.645,E2 -1201.645} C_VEL
LIN {X 0,Y 594.402,Z 332.441,A -85,B 0,C 180,E1 -1204.579,E2 -1204.579} C_VEL
LIN {X 0,Y 594.394,Z 332.441,A -85,B 0,C 180,E1 -1207.609,E2 -1207.609} C_VEL
LIN {X 0,Y 594.369,Z 332.445,A -85,B 0,C 180,E1 -1210.568,E2 -1210.568} C_VEL
LIN {X 0,Y 594.371,Z 332.448,A -85,B 0,C 180,E1 -1213.3,E2 -1213.3} C_VEL
LIN {X 0,Y 594.373,Z 332.442,A -85,B 0,C 180,E1 -1216.161,E2 -1216.161} C_VEL
LIN {X 0,Y 594.386,Z 332.443,A -85,B 0,C 180,E1 -1218.536,E2 -1218.536} C_VEL
LIN {X 0,Y 594.387,Z 332.444,A -85,B 0,C 180,E1 -1221.296,E2 -1221.296} C_VEL
LIN {X 0,Y 594.356,Z 332.444,A -85,B 0,C 180,E1 -1223.756,E2 -1223.756} C_VEL
LIN {X 0,Y 594.381,Z 332.442,A -85,B 0,C 180,E1 -1226.239,E2 -1226.239} C_VEL
LIN {X 0,Y 594.375,Z 332.448,A -85,B 0,C 180,E1 -1228.65,E2 -1228.65} C_VEL
LIN {X 0,Y 594.388,Z 332.447,A -85,B 0,C 180,E1 -1231.042,E2 -1231.042} C_VEL
LIN {X 0,Y 594.387,Z 332.44,A -85,B 0,C 180,E1 -1233.978,E2 -1233.978} C_VEL
LIN {X 0,Y 594.388,Z 332.442,A -85,B 0,C 180,E1 -1236.296,E2 -1236.296} C_VEL
LIN {X 0,Y 594.408,Z 332.441,A -85,B 0,C 180,E1 -1239.224,E2 -1239.224} C_VEL
LIN {X 0,Y 594.351,Z 332.446,A -85,B 0,C 180,E1 -1242.095,E2 -1242.095} C_VEL
LIN {X 0,Y 594.382,Z 332.604,A -85,B 0,C 180,E1 -1244.175,E2 -1244.175} C_VEL
LIN {X 0,Y 594.362,Z 345.366,A -85,B 0,C 180,E1 -1246.734,E2 -1246.734} C_VEL
LIN {X 0,Y 594.785,Z 350.161,A -85,B 0,C 180,E1 -1246.809,E2 -1246.809} C_VEL
LIN {X 0,Y 594.683,Z 450.859,A -85,B 0,C 180,E1 -1248.042,E2 -1248.042} C_VEL
LIN {X 0,Y 594.635,Z 464.172,A -85,B 0,C 180,E1 -1248.344,E2 -1248.344} C_VEL
LIN {X 0,Y 594.568,Z 476.012,A -85,B 0,C 180,E1 -1248.742,E2 -1248.742} C_VEL
LIN {X 0,Y 594.554,Z 487.742,A -85,B 0,C 180,E1 -1249.27,E2 -1249.27} C_VEL
LIN {X 0,Y 594.454,Z 499.516,A -85,B 0,C 180,E1 -1249.957,E2 -1249.957} C_VEL
LIN {X 0,Y 594.414,Z 510.022,A -85,B 0,C 180,E1 -1250.73,E2 -1250.73} C_VEL
LIN {X 0,Y 594.384,Z 518.643,A -85,B 0,C 180,E1 -1251.5,E2 -1251.5} C_VEL
LIN {X 0,Y 594.347,Z 526.578,A -85,B 0,C 180,E1 -1252.355,E2 -1252.355} C_VEL
LIN {X 0,Y 594.306,Z 534.383,A -85,B 0,C 180,E1 -1253.39,E2 -1253.39} C_VEL
LIN {X 0,Y 594.303,Z 539.596,A -85,B 0,C 180,E1 -1254.231,E2 -1254.231} C_VEL
LIN {X 0,Y 594.24,Z 544.744,A -85,B 0,C 180,E1 -1255.251,E2 -1255.251} C_VEL
LIN {X 0,Y 594.289,Z 548.742,A -85,B 0,C 180,E1 -1256.271,E2 -1256.271} C_VEL
LIN {X 0,Y 594.225,Z 551.696,A -85,B 0,C 180,E1 -1257.288,E2 -1257.288} C_VEL
LIN {X 0,Y 594.24,Z 553.13,A -85,B 0,C 180,E1 -1257.967,E2 -1257.967} C_VEL
LIN {X 0,Y 594.24,Z 554.757,A -85,B 0,C 180,E1 -1259.322,E2 -1259.322} C_VEL
LIN {X 0,Y 594.236,Z 554.996,A -85,B 0,C 180,E1 -1260,E2 -1260} C_VEL
LIN {X 0,Y 594.24,Z 554.817,A -85,B 0,C 180,E1 -1260.678,E2 -1260.678} C_VEL
LIN {X 0,Y 594.239,Z 553.279,A -85,B 0,C 180,E1 -1262.033,E2 -1262.033} C_VEL
LIN {X 0,Y 594.226,Z 551.913,A -85,B 0,C 180,E1 -1262.712,E2 -1262.712} C_VEL
LIN {X 0,Y 594.289,Z 549.042,A -85,B 0,C 180,E1 -1263.729,E2 -1263.729} C_VEL
LIN {X 0,Y 594.242,Z 545.145,A -85,B 0,C 180,E1 -1264.749,E2 -1264.749} C_VEL
LIN {X 0,Y 594.299,Z 540.104,A -85,B 0,C 180,E1 -1265.769,E2 -1265.769} C_VEL
LIN {X 0,Y 594.317,Z 533.771,A -85,B 0,C 180,E1 -1266.791,E2 -1266.791} C_VEL
LIN {X 0,Y 594.347,Z 525.876,A -85,B 0,C 180,E1 -1267.816,E2 -1267.816} C_VEL
LIN {X 0,Y 594.366,Z 517.803,A -85,B 0,C 180,E1 -1268.671,E2 -1268.671} C_VEL
LIN {X 0,Y 594.414,Z 507.947,A -85,B 0,C 180,E1 -1269.528,E2 -1269.528} C_VEL
LIN {X 0,Y 594.465,Z 496.912,A -85,B 0,C 180,E1 -1270.301,E2 -1270.301} C_VEL
LIN {X 0,Y 594.535,Z 486.075,A -85,B 0,C 180,E1 -1270.902,E2 -1270.902} C_VEL
LIN {X 0,Y 594.581,Z 475.636,A -85,B 0,C 180,E1 -1271.362,E2 -1271.362} C_VEL
LIN {X 0,Y 594.622,Z 462.785,A -85,B 0,C 180,E1 -1271.786,E2 -1271.786} C_VEL
LIN {X 0,Y 594.631,Z 461.725,A -85,B 0,C 180,E1 -1271.813,E2 -1271.813} C_VEL
LIN {X 0,Y 594.069,Z 456.04,A -85,B 0,C 180,E1 -1271.96,E2 -1271.96} C_VEL
LIN {X 0,Y 588.875,Z 439.363,A -85,B 0,C 180,E1 -1272.326,E2 -1272.326} C_VEL
LIN {X 0,Y 587.854,Z 433.61,A -85,B 0,C 180,E1 -1272.416,E2 -1272.416} C_VEL
LIN {X 0,Y 587.779,Z 431.657,A -85,B 0,C 180,E1 -1272.441,E2 -1272.441} C_VEL
LIN {X 0,Y 587.685,Z 347.583,A -85,B 0,C 180,E1 -1273.476,E2 -1273.476} C_VEL
LIN {X 0,Y 587.308,Z 345.27,A -85,B 0,C 180,E1 -1273.538,E2 -1273.538} C_VEL
LIN {X 0,Y 587.343,Z 333.321,A -85,B 0,C 180,E1 -1275.975,E2 -1275.975} C_VEL
LIN {X 0,Y 587.35,Z 333.32,A -85,B 0,C 180,E1 -1278.849,E2 -1278.849} C_VEL
LIN {X 0,Y 587.326,Z 333.323,A -85,B 0,C 180,E1 -1281.774,E2 -1281.774} C_VEL
LIN {X 0,Y 587.355,Z 333.319,A -85,B 0,C 180,E1 -1284.758,E2 -1284.758} C_VEL
LIN {X 0,Y 587.356,Z 333.319,A -85,B 0,C 180,E1 -1287.693,E2 -1287.693} C_VEL
LIN {X 0,Y 587.34,Z 333.319,A -85,B 0,C 180,E1 -1290.509,E2 -1290.509} C_VEL
LIN {X 0,Y 587.338,Z 333.325,A -85,B 0,C 180,E1 -1293.396,E2 -1293.396} C_VEL
LIN {X 0,Y 587.295,Z 333.324,A -85,B 0,C 180,E1 -1295.9,E2 -1295.9} C_VEL
LIN {X 0,Y 587.333,Z 333.32,A -85,B 0,C 180,E1 -1298.479,E2 -1298.479} C_VEL
LIN {X 0,Y 587.34,Z 333.327,A -85,B 0,C 180,E1 -1301.157,E2 -1301.157} C_VEL
LIN {X 0,Y 587.331,Z 333.319,A -85,B 0,C 180,E1 -1304.113,E2 -1304.113} C_VEL
LIN {X 0,Y 587.318,Z 333.331,A -85,B 0,C 180,E1 -1306.993,E2 -1306.993} C_VEL
LIN {X 0,Y 587.32,Z 333.321,A -85,B 0,C 180,E1 -1309.745,E2 -1309.745} C_VEL
LIN {X 0,Y 587.349,Z 333.319,A -85,B 0,C 180,E1 -1312.392,E2 -1312.392} C_VEL
LIN {X 0,Y 587.37,Z 333.314,A -85,B 0,C 180,E1 -1315.78,E2 -1315.78} C_VEL
LIN {X 0,Y 587.355,Z 333.317,A -85,B 0,C 180,E1 -1318.231,E2 -1318.231} C_VEL
LIN {X 0,Y 587.354,Z 333.326,A -85,B 0,C 180,E1 -1320.866,E2 -1320.866} C_VEL
LIN {X 0,Y 587.364,Z 333.315,A -85,B 0,C 180,E1 -1323.818,E2 -1323.818} C_VEL
LIN {X 0,Y 587.339,Z 333.318,A -85,B 0,C 180,E1 -1325.993,E2 -1325.993} C_VEL
LIN {X 0,Y 587.323,Z 333.322,A -85,B 0,C 180,E1 -1328.225,E2 -1328.225} C_VEL
LIN {X 0,Y 587.352,Z 333.32,A -85,B 0,C 180,E1 -1331.151,E2 -1331.151} C_VEL
LIN {X 0,Y 587.348,Z 333.319,A -85,B 0,C 180,E1 -1333.31,E2 -1333.31} C_VEL
LIN {X 0,Y 587.366,Z 333.317,A -85,B 0,C 180,E1 -1336.154,E2 -1336.154} C_VEL
LIN {X 0,Y 587.343,Z 333.323,A -85,B 0,C 180,E1 -1338.962,E2 -1338.962} C_VEL
LIN {X 0,Y 587.368,Z 333.314,A -85,B 0,C 180,E1 -1341.744,E2 -1341.744} C_VEL
LIN {X 0,Y 587.37,Z 333.323,A -85,B 0,C 180,E1 -1344.506,E2 -1344.506} C_VEL
LIN {X 0,Y 587.372,Z 333.315,A -85,B 0,C 180,E1 -1347.256,E2 -1347.256} C_VEL
LIN {X 0,Y 587.386,Z 333.314,A -85,B 0,C 180,E1 -1349.999,E2 -1349.999} C_VEL
LIN {X 0,Y 587.381,Z 333.319,A -85,B 0,C 180,E1 -1352.742,E2 -1352.742} C_VEL
LIN {X 0,Y 587.363,Z 333.315,A -85,B 0,C 180,E1 -1355.492,E2 -1355.492} C_VEL
LIN {X 0,Y 587.372,Z 333.321,A -85,B 0,C 180,E1 -1358.254,E2 -1358.254} C_VEL
LIN {X 0,Y 587.349,Z 333.317,A -85,B 0,C 180,E1 -1361.133,E2 -1361.133} C_VEL
LIN {X 0,Y 587.366,Z 333.323,A -85,B 0,C 180,E1 -1364.26,E2 -1364.26} C_VEL
LIN {X 0,Y 587.358,Z 333.315,A -85,B 0,C 180,E1 -1367.405,E2 -1367.405} C_VEL
LIN {X 0,Y 587.333,Z 333.329,A -85,B 0,C 180,E1 -1370.304,E2 -1370.304} C_VEL
LIN {X 0,Y 587.323,Z 333.32,A -85,B 0,C 180,E1 -1373.258,E2 -1373.258} C_VEL
LIN {X 0,Y 587.336,Z 333.319,A -85,B 0,C 180,E1 -1375.515,E2 -1375.515} C_VEL
LIN {X 0,Y 587.348,Z 333.32,A -85,B 0,C 180,E1 -1377.817,E2 -1377.817} C_VEL
LIN {X 0,Y 587.35,Z 333.321,A -85,B 0,C 180,E1 -1380.512,E2 -1380.512} C_VEL
LIN {X 0,Y 587.333,Z 333.319,A -85,B 0,C 180,E1 -1383.396,E2 -1383.396} C_VEL
LIN {X 0,Y 587.354,Z 333.322,A -85,B 0,C 180,E1 -1385.894,E2 -1385.894} C_VEL
LIN {X 0,Y 587.332,Z 333.323,A -85,B 0,C 180,E1 -1388.478,E2 -1388.478} C_VEL
LIN {X 0,Y 587.335,Z 333.318,A -85,B 0,C 180,E1 -1391.156,E2 -1391.156} C_VEL
LIN {X 0,Y 587.329,Z 333.328,A -85,B 0,C 180,E1 -1394.113,E2 -1394.113} C_VEL
LIN {X 0,Y 587.33,Z 333.319,A -85,B 0,C 180,E1 -1396.995,E2 -1396.995} C_VEL
LIN {X 0,Y 587.323,Z 333.326,A -85,B 0,C 180,E1 -1399.746,E2 -1399.746} C_VEL
LIN {X 0,Y 587.341,Z 333.321,A -85,B 0,C 180,E1 -1402.392,E2 -1402.392} C_VEL
LIN {X 0,Y 587.342,Z 333.317,A -85,B 0,C 180,E1 -1404.945,E2 -1404.945} C_VEL
LIN {X 0,Y 587.335,Z 333.321,A -85,B 0,C 180,E1 -1407.421,E2 -1407.421} C_VEL
LIN {X 0,Y 587.34,Z 333.328,A -85,B 0,C 180,E1 -1409.83,E2 -1409.83} C_VEL
LIN {X 0,Y 587.343,Z 333.32,A -85,B 0,C 180,E1 -1412.306,E2 -1412.306} C_VEL
LIN {X 0,Y 587.332,Z 333.32,A -85,B 0,C 180,E1 -1414.483,E2 -1414.483} C_VEL
LIN {X 0,Y 587.312,Z 333.322,A -85,B 0,C 180,E1 -1417.13,E2 -1417.13} C_VEL
LIN {X 0,Y 587.328,Z 333.329,A -85,B 0,C 180,E1 -1419.695,E2 -1419.695} C_VEL
LIN {X 0,Y 587.352,Z 333.316,A -85,B 0,C 180,E1 -1422.594,E2 -1422.594} C_VEL
LIN {X 0,Y 587.356,Z 333.325,A -85,B 0,C 180,E1 -1425.739,E2 -1425.739} C_VEL
LIN {X 0,Y 587.353,Z 333.316,A -85,B 0,C 180,E1 -1428.859,E2 -1428.859} C_VEL
LIN {X 0,Y 587.364,Z 333.323,A -85,B 0,C 180,E1 -1431.745,E2 -1431.745} C_VEL
LIN {X 0,Y 587.352,Z 333.316,A -85,B 0,C 180,E1 -1434.507,E2 -1434.507} C_VEL
LIN {X 0,Y 587.373,Z 333.319,A -85,B 0,C 180,E1 -1437.257,E2 -1437.257} C_VEL
LIN {X 0,Y 587.374,Z 333.316,A -85,B 0,C 180,E1 -1440,E2 -1440} C_VEL
LIN {X 0,Y 587.373,Z 333.314,A -85,B 0,C 180,E1 -1442.743,E2 -1442.743} C_VEL
LIN {X 0,Y 587.352,Z 333.326,A -85,B 0,C 180,E1 -1445.493,E2 -1445.493} C_VEL
LIN {X 0,Y 587.363,Z 333.315,A -85,B 0,C 180,E1 -1448.255,E2 -1448.255} C_VEL
LIN {X 0,Y 587.353,Z 333.322,A -85,B 0,C 180,E1 -1451.142,E2 -1451.142} C_VEL
LIN {X 0,Y 587.356,Z 333.316,A -85,B 0,C 180,E1 -1454.261,E2 -1454.261} C_VEL
LIN {X 0,Y 587.353,Z 333.325,A -85,B 0,C 180,E1 -1457.406,E2 -1457.406} C_VEL
LIN {X 0,Y 587.327,Z 333.319,A -85,B 0,C 180,E1 -1460.305,E2 -1460.305} C_VEL
LIN {X 0,Y 587.316,Z 333.331,A -85,B 0,C 180,E1 -1463.259,E2 -1463.259} C_VEL
LIN {X 0,Y 587.331,Z 333.324,A -85,B 0,C 180,E1 -1465.517,E2 -1465.517} C_VEL
LIN {X 0,Y 587.342,Z 333.319,A -85,B 0,C 180,E1 -1467.818,E2 -1467.818} C_VEL
LIN {X 0,Y 587.335,Z 333.319,A -85,B 0,C 180,E1 -1470.512,E2 -1470.512} C_VEL
LIN {X 0,Y 587.335,Z 333.328,A -85,B 0,C 180,E1 -1473.113,E2 -1473.113} C_VEL
LIN {X 0,Y 587.35,Z 333.317,A -85,B 0,C 180,E1 -1475.896,E2 -1475.896} C_VEL
LIN {X 0,Y 587.329,Z 333.32,A -85,B 0,C 180,E1 -1478.48,E2 -1478.48} C_VEL
LIN {X 0,Y 587.358,Z 333.324,A -85,B 0,C 180,E1 -1481.155,E2 -1481.155} C_VEL
LIN {X 0,Y 587.329,Z 333.319,A -85,B 0,C 180,E1 -1484.115,E2 -1484.115} C_VEL
LIN {X 0,Y 587.318,Z 333.331,A -85,B 0,C 180,E1 -1486.995,E2 -1486.995} C_VEL
LIN {X 0,Y 587.317,Z 333.321,A -85,B 0,C 180,E1 -1489.747,E2 -1489.747} C_VEL
LIN {X 0,Y 587.343,Z 333.319,A -85,B 0,C 180,E1 -1492.394,E2 -1492.394} C_VEL
LIN {X 0,Y 587.351,Z 333.326,A -85,B 0,C 180,E1 -1494.947,E2 -1494.947} C_VEL
LIN {X 0,Y 587.337,Z 333.32,A -85,B 0,C 180,E1 -1497.422,E2 -1497.422} C_VEL
LIN {X 0,Y 587.346,Z 333.317,A -85,B 0,C 180,E1 -1499.832,E2 -1499.832} C_VEL
LIN {X 0,Y 587.35,Z 333.32,A -85,B 0,C 180,E1 -1502.308,E2 -1502.308} C_VEL
LIN {X 0,Y 587.338,Z 333.325,A -85,B 0,C 180,E1 -1504.485,E2 -1504.485} C_VEL
LIN {X 0,Y 587.336,Z 333.405,A -85,B 0,C 180,E1 -1505.274,E2 -1505.274} C_VEL
LIN {X 0,Y 588.057,Z 337.636,A -85,B 0,C 180,E1 -1505.861,E2 -1505.861} C_VEL
LIN {X 0,Y 587.893,Z 359.128,A -85,B 0,C 180,E1 -1508.635,E2 -1508.635} C_VEL
LIN {X 0,Y 587.71,Z 381.952,A -85,B 0,C 180,E1 -1511.526,E2 -1511.526} C_VEL
LIN {X 0,Y 587.553,Z 404.912,A -85,B 0,C 180,E1 -1514.388,E2 -1514.388} C_VEL
LIN {X 0,Y 587.468,Z 421.953,A -85,B 0,C 180,E1 -1516.488,E2 -1516.488} C_VEL
LIN {X 0,Y 587.882,Z 426.794,A -85,B 0,C 180,E1 -1516.564,E2 -1516.564} C_VEL
LIN {X 0,Y 587.745,Z 530.994,A -85,B 0,C 180,E1 -1517.856,E2 -1517.856} C_VEL
LIN {X 0,Y 587.667,Z 544.25,A -85,B 0,C 180,E1 -1518.161,E2 -1518.161} C_VEL
LIN {X 0,Y 587.605,Z 556.641,A -85,B 0,C 180,E1 -1518.585,E2 -1518.585} C_VEL
LIN {X 0,Y 587.552,Z 568.647,A -85,B 0,C 180,E1 -1519.142,E2 -1519.142} C_VEL
LIN {X 0,Y 587.465,Z 580.214,A -85,B 0,C 180,E1 -1519.837,E2 -1519.837} C_VEL
LIN {X 0,Y 587.391,Z 590.608,A -85,B 0,C 180,E1 -1520.619,E2 -1520.619} C_VEL
LIN {X 0,Y 587.321,Z 599.121,A -85,B 0,C 180,E1 -1521.398,E2 -1521.398} C_VEL
LIN {X 0,Y 587.273,Z 606.968,A -85,B 0,C 180,E1 -1522.264,E2 -1522.264} C_VEL
LIN {X 0,Y 587.232,Z 613.475,A -85,B 0,C 180,E1 -1523.127,E2 -1523.127} C_VEL
LIN {X 0,Y 587.236,Z 619.871,A -85,B 0,C 180,E1 -1524.162,E2 -1524.162} C_VEL
LIN {X 0,Y 587.147,Z 624.953,A -85,B 0,C 180,E1 -1525.194,E2 -1525.194} C_VEL
LIN {X 0,Y 587.212,Z 628.898,A -85,B 0,C 180,E1 -1526.227,E2 -1526.227} C_VEL
LIN {X 0,Y 587.132,Z 631.811,A -85,B 0,C 180,E1 -1527.256,E2 -1527.256} C_VEL
LIN {X 0,Y 587.139,Z 633.202,A -85,B 0,C 180,E1 -1527.943,E2 -1527.943} C_VEL
LIN {X 0,Y 587.14,Z 634.785,A -85,B 0,C 180,E1 -1529.315,E2 -1529.315} C_VEL
LIN {X 0,Y 587.137,Z 635,A -85,B 0,C 180,E1 -1530.001,E2 -1530.001} C_VEL
LIN {X 0,Y 587.147,Z 634.184,A -85,B 0,C 180,E1 -1531.373,E2 -1531.373} C_VEL
LIN {X 0,Y 587.139,Z 633.2,A -85,B 0,C 180,E1 -1532.059,E2 -1532.059} C_VEL
LIN {X 0,Y 587.132,Z 631.808,A -85,B 0,C 180,E1 -1532.745,E2 -1532.745} C_VEL
LIN {X 0,Y 587.212,Z 628.893,A -85,B 0,C 180,E1 -1533.775,E2 -1533.775} C_VEL
LIN {X 0,Y 587.147,Z 624.946,A -85,B 0,C 180,E1 -1534.807,E2 -1534.807} C_VEL
LIN {X 0,Y 587.217,Z 618.873,A -85,B 0,C 180,E1 -1536.012,E2 -1536.012} C_VEL
LIN {X 0,Y 587.246,Z 612.231,A -85,B 0,C 180,E1 -1537.047,E2 -1537.047} C_VEL
LIN {X 0,Y 587.3,Z 603.984,A -85,B 0,C 180,E1 -1538.084,E2 -1538.084} C_VEL
LIN {X 0,Y 587.344,Z 595.53,A -85,B 0,C 180,E1 -1538.95,E2 -1538.95} C_VEL
LIN {X 0,Y 587.416,Z 585.086,A -85,B 0,C 180,E1 -1539.817,E2 -1539.817} C_VEL
LIN {X 0,Y 587.496,Z 574.746,A -85,B 0,C 180,E1 -1540.512,E2 -1540.512} C_VEL
LIN {X 0,Y 587.585,Z 562.795,A -85,B 0,C 180,E1 -1541.149,E2 -1541.149} C_VEL
LIN {X 0,Y 587.628,Z 550.574,A -85,B 0,C 180,E1 -1541.64,E2 -1541.64} C_VEL
LIN {X 0,Y 587.711,Z 537.406,A -85,B 0,C 180,E1 -1542.015,E2 -1542.015} C_VEL
LIN {X 0,Y 587.773,Z 525.03,A -85,B 0,C 180,E1 -1542.232,E2 -1542.232} C_VEL
LIN {X 0,Y 587.752,Z 424.091,A -85,B 0,C 180,E1 -1543.472,E2 -1543.472} C_VEL
LIN {X 0,Y 587.469,Z 421.94,A -85,B 0,C 180,E1 -1543.513,E2 -1543.513} C_VEL
LIN {X 0,Y 587.591,Z 397.724,A -85,B 0,C 180,E1 -1546.504,E2 -1546.504} C_VEL
LIN {X 0,Y 587.746,Z 375.439,A -85,B 0,C 180,E1 -1549.295,E2 -1549.295} C_VEL
LIN {X 0,Y 587.941,Z 353.238,A -85,B 0,C 180,E1 -1552.12,E2 -1552.12} C_VEL
LIN {X 0,Y 588.016,Z 336.361,A -85,B 0,C 180,E1 -1554.308,E2 -1554.308} C_VEL
LIN {X 0,Y 587.317,Z 333.329,A -85,B 0,C 180,E1 -1554.761,E2 -1554.761} C_VEL
LIN {X 0,Y 587.335,Z 333.328,A -85,B 0,C 180,E1 -1557.047,E2 -1557.047} C_VEL
LIN {X 0,Y 587.353,Z 333.323,A -85,B 0,C 180,E1 -1559.38,E2 -1559.38} C_VEL
LIN {X 0,Y 587.358,Z 333.317,A -85,B 0,C 180,E1 -1561.837,E2 -1561.837} C_VEL
LIN {X 0,Y 587.36,Z 333.316,A -85,B 0,C 180,E1 -1564.349,E2 -1564.349} C_VEL
LIN {X 0,Y 587.35,Z 333.319,A -85,B 0,C 180,E1 -1567.608,E2 -1567.608} C_VEL
LIN {X 0,Y 587.321,Z 333.321,A -85,B 0,C 180,E1 -1570.254,E2 -1570.254} C_VEL
LIN {X 0,Y 587.32,Z 333.329,A -85,B 0,C 180,E1 -1573.118,E2 -1573.118} C_VEL
LIN {X 0,Y 587.329,Z 333.319,A -85,B 0,C 180,E1 -1576.05,E2 -1576.05} C_VEL
LIN {X 0,Y 587.342,Z 333.327,A -85,B 0,C 180,E1 -1578.925,E2 -1578.925} C_VEL
LIN {X 0,Y 587.334,Z 333.32,A -85,B 0,C 180,E1 -1581.521,E2 -1581.521} C_VEL
LIN {X 0,Y 587.296,Z 333.323,A -85,B 0,C 180,E1 -1584.1,E2 -1584.1} C_VEL
LIN {X 0,Y 587.338,Z 333.323,A -85,B 0,C 180,E1 -1586.603,E2 -1586.603} C_VEL
LIN {X 0,Y 587.341,Z 333.319,A -85,B 0,C 180,E1 -1589.49,E2 -1589.49} C_VEL
LIN {X 0,Y 587.357,Z 333.318,A -85,B 0,C 180,E1 -1592.307,E2 -1592.307} C_VEL
LIN {X 0,Y 587.355,Z 333.32,A -85,B 0,C 180,E1 -1595.241,E2 -1595.241} C_VEL
LIN {X 0,Y 587.327,Z 333.322,A -85,B 0,C 180,E1 -1598.226,E2 -1598.226} C_VEL
LIN {X 0,Y 587.352,Z 333.321,A -85,B 0,C 180,E1 -1601.151,E2 -1601.151} C_VEL
LIN {X 0,Y 587.343,Z 333.32,A -85,B 0,C 180,E1 -1604.025,E2 -1604.025} C_VEL
LIN {X 0,Y 587.345,Z 333.698,A -85,B 0,C 180,E1 -1604.203,E2 -1604.203} C_VEL
LIN {X 0,Y 587.333,Z 345.369,A -85,B 0,C 180,E1 -1606.572,E2 -1606.572} C_VEL
LIN {X 0,Y 587.876,Z 350.206,A -85,B 0,C 180,E1 -1606.651,E2 -1606.651} C_VEL
LIN {X 0,Y 587.74,Z 450.89,A -85,B 0,C 180,E1 -1607.899,E2 -1607.899} C_VEL
LIN {X 0,Y 587.704,Z 464.2,A -85,B 0,C 180,E1 -1608.205,E2 -1608.205} C_VEL
LIN {X 0,Y 587.597,Z 476.66,A -85,B 0,C 180,E1 -1608.633,E2 -1608.633} C_VEL
LIN {X 0,Y 587.572,Z 487.749,A -85,B 0,C 180,E1 -1609.141,E2 -1609.141} C_VEL
LIN {X 0,Y 587.428,Z 499.521,A -85,B 0,C 180,E1 -1609.836,E2 -1609.836} C_VEL
LIN {X 0,Y 587.393,Z 510.024,A -85,B 0,C 180,E1 -1610.618,E2 -1610.618} C_VEL
LIN {X 0,Y 587.323,Z 518.648,A -85,B 0,C 180,E1 -1611.397,E2 -1611.397} C_VEL
LIN {X 0,Y 587.272,Z 527.964,A -85,B 0,C 180,E1 -1612.436,E2 -1612.436} C_VEL
LIN {X 0,Y 587.247,Z 534.816,A -85,B 0,C 180,E1 -1613.376,E2 -1613.376} C_VEL
LIN {X 0,Y 587.211,Z 541.447,A -85,B 0,C 180,E1 -1614.506,E2 -1614.506} C_VEL
LIN {X 0,Y 587.188,Z 546.193,A -85,B 0,C 180,E1 -1615.538,E2 -1615.538} C_VEL
LIN {X 0,Y 587.195,Z 549.822,A -85,B 0,C 180,E1 -1616.569,E2 -1616.569} C_VEL
LIN {X 0,Y 587.132,Z 551.699,A -85,B 0,C 180,E1 -1617.256,E2 -1617.256} C_VEL
LIN {X 0,Y 587.139,Z 553.128,A -85,B 0,C 180,E1 -1617.942,E2 -1617.942} C_VEL
LIN {X 0,Y 587.14,Z 554.759,A -85,B 0,C 180,E1 -1619.314,E2 -1619.314} C_VEL
LIN {X 0,Y 587.137,Z 554.996,A -85,B 0,C 180,E1 -1620,E2 -1620} C_VEL
LIN {X 0,Y 587.14,Z 554.814,A -85,B 0,C 180,E1 -1620.686,E2 -1620.686} C_VEL
LIN {X 0,Y 587.138,Z 553.28,A -85,B 0,C 180,E1 -1622.058,E2 -1622.058} C_VEL
LIN {X 0,Y 587.133,Z 551.91,A -85,B 0,C 180,E1 -1622.744,E2 -1622.744} C_VEL
LIN {X 0,Y 587.213,Z 549.042,A -85,B 0,C 180,E1 -1623.774,E2 -1623.774} C_VEL
LIN {X 0,Y 587.147,Z 545.144,A -85,B 0,C 180,E1 -1624.806,E2 -1624.806} C_VEL
LIN {X 0,Y 587.229,Z 540.093,A -85,B 0,C 180,E1 -1625.839,E2 -1625.839} C_VEL
LIN {X 0,Y 587.23,Z 533.76,A -85,B 0,C 180,E1 -1626.874,E2 -1626.874} C_VEL
LIN {X 0,Y 587.288,Z 525.874,A -85,B 0,C 180,E1 -1627.91,E2 -1627.91} C_VEL
LIN {X 0,Y 587.324,Z 517.797,A -85,B 0,C 180,E1 -1628.776,E2 -1628.776} C_VEL
LIN {X 0,Y 587.383,Z 507.93,A -85,B 0,C 180,E1 -1629.643,E2 -1629.643} C_VEL
LIN {X 0,Y 587.484,Z 496.906,A -85,B 0,C 180,E1 -1630.424,E2 -1630.424} C_VEL
LIN {X 0,Y 587.543,Z 486.06,A -85,B 0,C 180,E1 -1631.034,E2 -1631.034} C_VEL
LIN {X 0,Y 587.614,Z 474.271,A -85,B 0,C 180,E1 -1631.551,E2 -1631.551} C_VEL
LIN {X 0,Y 587.7,Z 461.102,A -85,B 0,C 180,E1 -1631.97,E2 -1631.97} C_VEL
LIN {X 0,Y 587.777,Z 448.188,A -85,B 0,C 180,E1 -1632.231,E2 -1632.231} C_VEL
LIN {X 0,Y 587.779,Z 431.657,A -85,B 0,C 180,E1 -1632.441,E2 -1632.441} C_VEL
LIN {X 0,Y 587.161,Z 425.85,A -85,B 0,C 180,E1 -1632.526,E2 -1632.526} C_VEL
LIN {X 0,Y 581.607,Z 407.152,A -85,B 0,C 180,E1 -1632.879,E2 -1632.879} C_VEL
LIN {X 0,Y 580.929,Z 401.345,A -85,B 0,C 180,E1 -1632.966,E2 -1632.966} C_VEL
LIN {X 0,Y 580.9,Z 348.994,A -85,B 0,C 180,E1 -1633.618,E2 -1633.618} C_VEL
LIN {X 0,Y 580.274,Z 345.267,A -85,B 0,C 180,E1 -1633.705,E2 -1633.705} C_VEL
LIN {X 0,Y 580.298,Z 334.199,A -85,B 0,C 180,E1 -1635.993,E2 -1635.993} C_VEL
LIN {X 0,Y 580.264,Z 334.2,A -85,B 0,C 180,E1 -1638.355,E2 -1638.355} C_VEL
LIN {X 0,Y 580.305,Z 334.202,A -85,B 0,C 180,E1 -1641.165,E2 -1641.165} C_VEL
LIN {X 0,Y 580.281,Z 334.203,A -85,B 0,C 180,E1 -1643.558,E2 -1643.558} C_VEL
LIN {X 0,Y 580.294,Z 334.198,A -85,B 0,C 180,E1 -1645.849,E2 -1645.849} C_VEL
LIN {X 0,Y 580.303,Z 334.195,A -85,B 0,C 180,E1 -1648.185,E2 -1648.185} C_VEL
LIN {X 0,Y 580.287,Z 334.199,A -85,B 0,C 180,E1 -1650.694,E2 -1650.694} C_VEL
LIN {X 0,Y 580.307,Z 334.202,A -85,B 0,C 180,E1 -1653.316,E2 -1653.316} C_VEL
LIN {X 0,Y 580.249,Z 334.203,A -85,B 0,C 180,E1 -1655.756,E2 -1655.756} C_VEL
LIN {X 0,Y 580.292,Z 334.196,A -85,B 0,C 180,E1 -1658.146,E2 -1658.146} C_VEL
LIN {X 0,Y 580.302,Z 334.201,A -85,B 0,C 180,E1 -1660.843,E2 -1660.843} C_VEL
LIN {X 0,Y 580.284,Z 334.199,A -85,B 0,C 180,E1 -1663.657,E2 -1663.657} C_VEL
LIN {X 0,Y 580.281,Z 334.201,A -85,B 0,C 180,E1 -1666.609,E2 -1666.609} C_VEL
LIN {X 0,Y 580.303,Z 334.202,A -85,B 0,C 180,E1 -1669.156,E2 -1669.156} C_VEL
LIN {X 0,Y 580.294,Z 334.196,A -85,B 0,C 180,E1 -1671.927,E2 -1671.927} C_VEL
LIN {X 0,Y 580.262,Z 334.203,A -85,B 0,C 180,E1 -1674.453,E2 -1674.453} C_VEL
LIN {X 0,Y 580.293,Z 334.205,A -85,B 0,C 180,E1 -1676.975,E2 -1676.975} C_VEL
LIN {X 0,Y 580.307,Z 334.196,A -85,B 0,C 180,E1 -1679.425,E2 -1679.425} C_VEL
LIN {X 0,Y 580.301,Z 334.196,A -85,B 0,C 180,E1 -1682.141,E2 -1682.141} C_VEL
LIN {X 0,Y 580.326,Z 334.195,A -85,B 0,C 180,E1 -1685.269,E2 -1685.269} C_VEL
LIN {X 0,Y 580.274,Z 334.198,A -85,B 0,C 180,E1 -1687.947,E2 -1687.947} C_VEL
LIN {X 0,Y 580.302,Z 334.202,A -85,B 0,C 180,E1 -1690.913,E2 -1690.913} C_VEL
LIN {X 0,Y 580.31,Z 334.198,A -85,B 0,C 180,E1 -1693.102,E2 -1693.102} C_VEL
LIN {X 0,Y 580.332,Z 334.192,A -85,B 0,C 180,E1 -1695.983,E2 -1695.983} C_VEL
LIN {X 0,Y 580.309,Z 334.201,A -85,B 0,C 180,E1 -1698.826,E2 -1698.826} C_VEL
LIN {X 0,Y 580.331,Z 334.191,A -85,B 0,C 180,E1 -1701.643,E2 -1701.643} C_VEL
LIN {X 0,Y 580.336,Z 334.198,A -85,B 0,C 180,E1 -1704.44,E2 -1704.44} C_VEL
LIN {X 0,Y 580.339,Z 334.191,A -85,B 0,C 180,E1 -1707.223,E2 -1707.223} C_VEL
LIN {X 0,Y 580.356,Z 334.19,A -85,B 0,C 180,E1 -1709.999,E2 -1709.999} C_VEL
LIN {X 0,Y 580.346,Z 334.195,A -85,B 0,C 180,E1 -1712.776,E2 -1712.776} C_VEL
LIN {X 0,Y 580.331,Z 334.191,A -85,B 0,C 180,E1 -1715.559,E2 -1715.559} C_VEL
LIN {X 0,Y 580.336,Z 334.199,A -85,B 0,C 180,E1 -1718.355,E2 -1718.355} C_VEL
LIN {X 0,Y 580.301,Z 334.195,A -85,B 0,C 180,E1 -1721.19,E2 -1721.19} C_VEL
LIN {X 0,Y 580.327,Z 334.196,A -85,B 0,C 180,E1 -1724.016,E2 -1724.016} C_VEL
LIN {X 0,Y 580.314,Z 334.195,A -85,B 0,C 180,E1 -1726.914,E2 -1726.914} C_VEL
LIN {X 0,Y 580.306,Z 334.197,A -85,B 0,C 180,E1 -1729.821,E2 -1729.821} C_VEL
LIN {X 0,Y 580.295,Z 334.198,A -85,B 0,C 180,E1 -1732.801,E2 -1732.801} C_VEL
LIN {X 0,Y 580.306,Z 334.194,A -85,B 0,C 180,E1 -1735.079,E2 -1735.079} C_VEL
LIN {X 0,Y 580.318,Z 334.197,A -85,B 0,C 180,E1 -1737.862,E2 -1737.862} C_VEL
LIN {X 0,Y 580.298,Z 334.198,A -85,B 0,C 180,E1 -1740.697,E2 -1740.697} C_VEL
LIN {X 0,Y 580.302,Z 334.195,A -85,B 0,C 180,E1 -1743.316,E2 -1743.316} C_VEL
LIN {X 0,Y 580.324,Z 334.196,A -85,B 0,C 180,E1 -1745.767,E2 -1745.767} C_VEL
LIN {X 0,Y 580.287,Z 334.206,A -85,B 0,C 180,E1 -1748.145,E2 -1748.145} C_VEL
LIN {X 0,Y 580.3,Z 334.195,A -85,B 0,C 180,E1 -1750.842,E2 -1750.842} C_VEL
LIN {X 0,Y 580.282,Z 334.201,A -85,B 0,C 180,E1 -1753.656,E2 -1753.656} C_VEL
LIN {X 0,Y 580.286,Z 334.198,A -85,B 0,C 180,E1 -1756.607,E2 -1756.607} C_VEL
LIN {X 0,Y 580.314,Z 334.193,A -85,B 0,C 180,E1 -1759.158,E2 -1759.158} C_VEL
LIN {X 0,Y 580.286,Z 334.207,A -85,B 0,C 180,E1 -1761.926,E2 -1761.926} C_VEL
LIN {X 0,Y 580.299,Z 334.197,A -85,B 0,C 180,E1 -1764.456,E2 -1764.456} C_VEL
LIN {X 0,Y 580.286,Z 334.196,A -85,B 0,C 180,E1 -1766.975,E2 -1766.975} C_VEL
LIN {X 0,Y 580.303,Z 334.198,A -85,B 0,C 180,E1 -1769.426,E2 -1769.426} C_VEL
LIN {X 0,Y 580.312,Z 334.198,A -85,B 0,C 180,E1 -1772.136,E2 -1772.136} C_VEL
LIN {X 0,Y 580.301,Z 334.195,A -85,B 0,C 180,E1 -1774.92,E2 -1774.92} C_VEL
LIN {X 0,Y 580.27,Z 334.206,A -85,B 0,C 180,E1 -1777.947,E2 -1777.947} C_VEL
LIN {X 0,Y 580.309,Z 334.194,A -85,B 0,C 180,E1 -1780.914,E2 -1780.914} C_VEL
LIN {X 0,Y 580.277,Z 334.206,A -85,B 0,C 180,E1 -1783.826,E2 -1783.826} C_VEL
LIN {X 0,Y 580.318,Z 334.197,A -85,B 0,C 180,E1 -1785.983,E2 -1785.983} C_VEL
LIN {X 0,Y 580.322,Z 334.192,A -85,B 0,C 180,E1 -1788.827,E2 -1788.827} C_VEL
LIN {X 0,Y 580.328,Z 334.201,A -85,B 0,C 180,E1 -1791.644,E2 -1791.644} C_VEL
LIN {X 0,Y 580.318,Z 334.192,A -85,B 0,C 180,E1 -1794.44,E2 -1794.44} C_VEL
LIN {X 0,Y 580.339,Z 334.194,A -85,B 0,C 180,E1 -1797.224,E2 -1797.224} C_VEL
LIN {X 0,Y 580.343,Z 334.192,A -85,B 0,C 180,E1 -1800,E2 -1800} C_VEL
LIN {X 0,Y 580.339,Z 334.19,A -85,B 0,C 180,E1 -1802.777,E2 -1802.777} C_VEL
LIN {X 0,Y 580.318,Z 334.201,A -85,B 0,C 180,E1 -1805.56,E2 -1805.56} C_VEL
LIN {X 0,Y 580.327,Z 334.191,A -85,B 0,C 180,E1 -1808.356,E2 -1808.356} C_VEL
LIN {X 0,Y 580.324,Z 334.198,A -85,B 0,C 180,E1 -1811.209,E2 -1811.209} C_VEL
LIN {X 0,Y 580.306,Z 334.194,A -85,B 0,C 180,E1 -1814.339,E2 -1814.339} C_VEL
LIN {X 0,Y 580.307,Z 334.197,A -85,B 0,C 180,E1 -1816.916,E2 -1816.916} C_VEL
LIN {X 0,Y 580.3,Z 334.197,A -85,B 0,C 180,E1 -1819.823,E2 -1819.823} C_VEL
LIN {X 0,Y 580.269,Z 334.199,A -85,B 0,C 180,E1 -1822.053,E2 -1822.053} C_VEL
LIN {X 0,Y 580.301,Z 334.202,A -85,B 0,C 180,E1 -1825.08,E2 -1825.08} C_VEL
LIN {X 0,Y 580.313,Z 334.194,A -85,B 0,C 180,E1 -1827.864,E2 -1827.864} C_VEL
LIN {X 0,Y 580.286,Z 334.199,A -85,B 0,C 180,E1 -1830.697,E2 -1830.697} C_VEL
LIN {X 0,Y 580.299,Z 334.202,A -85,B 0,C 180,E1 -1833.318,E2 -1833.318} C_VEL
LIN {X 0,Y 580.319,Z 334.193,A -85,B 0,C 180,E1 -1835.768,E2 -1835.768} C_VEL
LIN {X 0,Y 580.284,Z 334.197,A -85,B 0,C 180,E1 -1838.147,E2 -1838.147} C_VEL
LIN {X 0,Y 580.315,Z 334.199,A -85,B 0,C 180,E1 -1840.842,E2 -1840.842} C_VEL
LIN {X 0,Y 580.286,Z 334.198,A -85,B 0,C 180,E1 -1843.657,E2 -1843.657} C_VEL
LIN {X 0,Y 580.281,Z 334.201,A -85,B 0,C 180,E1 -1846.609,E2 -1846.609} C_VEL
LIN {X 0,Y 580.298,Z 334.202,A -85,B 0,C 180,E1 -1849.158,E2 -1849.158} C_VEL
LIN {X 0,Y 580.288,Z 334.196,A -85,B 0,C 180,E1 -1851.928,E2 -1851.928} C_VEL
LIN {X 0,Y 580.306,Z 334.197,A -85,B 0,C 180,E1 -1854.458,E2 -1854.458} C_VEL
LIN {X 0,Y 580.289,Z 334.205,A -85,B 0,C 180,E1 -1856.976,E2 -1856.976} C_VEL
LIN {X 0,Y 580.309,Z 334.196,A -85,B 0,C 180,E1 -1859.427,E2 -1859.427} C_VEL
LIN {X 0,Y 580.318,Z 334.195,A -85,B 0,C 180,E1 -1862.138,E2 -1862.138} C_VEL
LIN {X 0,Y 580.292,Z 334.206,A -85,B 0,C 180,E1 -1864.921,E2 -1864.921} C_VEL
LIN {X 0,Y 580.315,Z 334.385,A -85,B 0,C 180,E1 -1865.107,E2 -1865.107} C_VEL
LIN {X 0,Y 581.215,Z 338.9,A -85,B 0,C 180,E1 -1865.726,E2 -1865.726} C_VEL
LIN {X 0,Y 580.984,Z 360.572,A -85,B 0,C 180,E1 -1868.555,E2 -1868.555} C_VEL
LIN {X 0,Y 580.77,Z 383.387,A -85,B 0,C 180,E1 -1871.48,E2 -1871.48} C_VEL
LIN {X 0,Y 580.546,Z 406.347,A -85,B 0,C 180,E1 -1874.375,E2 -1874.375} C_VEL
LIN {X 0,Y 580.442,Z 421.953,A -85,B 0,C 180,E1 -1876.322,E2 -1876.322} C_VEL
LIN {X 0,Y 580.984,Z 426.794,A -85,B 0,C 180,E1 -1876.402,E2 -1876.402} C_VEL
LIN {X 0,Y 580.805,Z 530.994,A -85,B 0,C 180,E1 -1877.709,E2 -1877.709} C_VEL
LIN {X 0,Y 580.725,Z 544.251,A -85,B 0,C 180,E1 -1878.018,E2 -1878.018} C_VEL
LIN {X 0,Y 580.638,Z 557.496,A -85,B 0,C 180,E1 -1878.48,E2 -1878.48} C_VEL
LIN {X 0,Y 580.567,Z 568.646,A -85,B 0,C 180,E1 -1879.01,E2 -1879.01} C_VEL
LIN {X 0,Y 580.444,Z 580.216,A -85,B 0,C 180,E1 -1879.713,E2 -1879.713} C_VEL
LIN {X 0,Y 580.341,Z 590.61,A -85,B 0,C 180,E1 -1880.504,E2 -1880.504} C_VEL
LIN {X 0,Y 580.271,Z 599.121,A -85,B 0,C 180,E1 -1881.293,E2 -1881.293} C_VEL
LIN {X 0,Y 580.221,Z 606.968,A -85,B 0,C 180,E1 -1882.169,E2 -1882.169} C_VEL
LIN {X 0,Y 580.154,Z 614.655,A -85,B 0,C 180,E1 -1883.222,E2 -1883.222} C_VEL
LIN {X 0,Y 580.139,Z 621.685,A -85,B 0,C 180,E1 -1884.439,E2 -1884.439} C_VEL
LIN {X 0,Y 580.108,Z 626.375,A -85,B 0,C 180,E1 -1885.484,E2 -1885.484} C_VEL
LIN {X 0,Y 580.123,Z 629.959,A -85,B 0,C 180,E1 -1886.528,E2 -1886.528} C_VEL
LIN {X 0,Y 580.043,Z 631.81,A -85,B 0,C 180,E1 -1887.223,E2 -1887.223} C_VEL
LIN {X 0,Y 580.038,Z 633.201,A -85,B 0,C 180,E1 -1887.918,E2 -1887.918} C_VEL
LIN {X 0,Y 580.04,Z 634.785,A -85,B 0,C 180,E1 -1889.307,E2 -1889.307} C_VEL
LIN {X 0,Y 580.037,Z 635,A -85,B 0,C 180,E1 -1890.001,E2 -1890.001} C_VEL
LIN {X 0,Y 580.047,Z 634.185,A -85,B 0,C 180,E1 -1891.389,E2 -1891.389} C_VEL
LIN {X 0,Y 580.039,Z 633.199,A -85,B 0,C 180,E1 -1892.084,E2 -1892.084} C_VEL
LIN {X 0,Y 580.043,Z 631.808,A -85,B 0,C 180,E1 -1892.779,E2 -1892.779} C_VEL
LIN {X 0,Y 580.109,Z 628.893,A -85,B 0,C 180,E1 -1893.821,E2 -1893.821} C_VEL
LIN {X 0,Y 580.054,Z 624.946,A -85,B 0,C 180,E1 -1894.866,E2 -1894.866} C_VEL
LIN {X 0,Y 580.139,Z 618.873,A -85,B 0,C 180,E1 -1896.086,E2 -1896.086} C_VEL
LIN {X 0,Y 580.185,Z 612.232,A -85,B 0,C 180,E1 -1897.133,E2 -1897.133} C_VEL
LIN {X 0,Y 580.251,Z 603.984,A -85,B 0,C 180,E1 -1898.183,E2 -1898.183} C_VEL
LIN {X 0,Y 580.308,Z 595.53,A -85,B 0,C 180,E1 -1899.059,E2 -1899.059} C_VEL
LIN {X 0,Y 580.417,Z 585.087,A -85,B 0,C 180,E1 -1899.937,E2 -1899.937} C_VEL
LIN {X 0,Y 580.507,Z 574.744,A -85,B 0,C 180,E1 -1900.64,E2 -1900.64} C_VEL
LIN {X 0,Y 580.598,Z 563.227,A -85,B 0,C 180,E1 -1901.265,E2 -1901.265} C_VEL
LIN {X 0,Y 580.666,Z 550.45,A -85,B 0,C 180,E1 -1901.786,E2 -1901.786} C_VEL
LIN {X 0,Y 580.772,Z 537.405,A -85,B 0,C 180,E1 -1902.16,E2 -1902.16} C_VEL
LIN {X 0,Y 580.836,Z 525.03,A -85,B 0,C 180,E1 -1902.381,E2 -1902.381} C_VEL
LIN {X 0,Y 580.86,Z 424.871,A -85,B 0,C 180,E1 -1903.625,E2 -1903.625} C_VEL
LIN {X 0,Y 580.443,Z 421.94,A -85,B 0,C 180,E1 -1903.68,E2 -1903.68} C_VEL
LIN {X 0,Y 580.623,Z 399.159,A -85,B 0,C 180,E1 -1906.527,E2 -1906.527} C_VEL
LIN {X 0,Y 580.811,Z 377.307,A -85,B 0,C 180,E1 -1909.295,E2 -1909.295} C_VEL
LIN {X 0,Y 581.025,Z 356.108,A -85,B 0,C 180,E1 -1912.023,E2 -1912.023} C_VEL
LIN {X 0,Y 581.212,Z 338.887,A -85,B 0,C 180,E1 -1914.276,E2 -1914.276} C_VEL
LIN {X 0,Y 580.286,Z 334.206,A -85,B 0,C 180,E1 -1914.922,E2 -1914.922} C_VEL
LIN {X 0,Y 580.302,Z 334.197,A -85,B 0,C 180,E1 -1917.859,E2 -1917.859} C_VEL
LIN {X 0,Y 580.298,Z 334.199,A -85,B 0,C 180,E1 -1920.696,E2 -1920.696} C_VEL
LIN {X 0,Y 580.308,Z 334.202,A -85,B 0,C 180,E1 -1923.316,E2 -1923.316} C_VEL
LIN {X 0,Y 580.255,Z 334.202,A -85,B 0,C 180,E1 -1925.757,E2 -1925.757} C_VEL
LIN {X 0,Y 580.294,Z 334.196,A -85,B 0,C 180,E1 -1928.147,E2 -1928.147} C_VEL
LIN {X 0,Y 580.303,Z 334.201,A -85,B 0,C 180,E1 -1930.844,E2 -1930.844} C_VEL
LIN {X 0,Y 580.284,Z 334.198,A -85,B 0,C 180,E1 -1933.658,E2 -1933.658} C_VEL
LIN {X 0,Y 580.284,Z 334.201,A -85,B 0,C 180,E1 -1936.609,E2 -1936.609} C_VEL
LIN {X 0,Y 580.304,Z 334.202,A -85,B 0,C 180,E1 -1939.157,E2 -1939.157} C_VEL
LIN {X 0,Y 580.295,Z 334.196,A -85,B 0,C 180,E1 -1941.927,E2 -1941.927} C_VEL
LIN {X 0,Y 580.255,Z 334.203,A -85,B 0,C 180,E1 -1944.453,E2 -1944.453} C_VEL
LIN {X 0,Y 580.296,Z 334.204,A -85,B 0,C 180,E1 -1946.975,E2 -1946.975} C_VEL
LIN {X 0,Y 580.3,Z 334.197,A -85,B 0,C 180,E1 -1949.425,E2 -1949.425} C_VEL
LIN {X 0,Y 580.303,Z 334.196,A -85,B 0,C 180,E1 -1952.141,E2 -1952.141} C_VEL
LIN {X 0,Y 580.326,Z 334.195,A -85,B 0,C 180,E1 -1955.27,E2 -1955.27} C_VEL
LIN {X 0,Y 580.277,Z 334.199,A -85,B 0,C 180,E1 -1957.947,E2 -1957.947} C_VEL
LIN {X 0,Y 580.304,Z 334.203,A -85,B 0,C 180,E1 -1960.913,E2 -1960.913} C_VEL
LIN {X 0,Y 580.293,Z 334.199,A -85,B 0,C 180,E1 -1963.826,E2 -1963.826} C_VEL
LIN {X 0,Y 580.304,Z 334.355,A -85,B 0,C 180,E1 -1964.142,E2 -1964.142} C_VEL
LIN {X 0,Y 580.284,Z 345.372,A -85,B 0,C 180,E1 -1966.406,E2 -1966.406} C_VEL
LIN {X 0,Y 580.987,Z 350.252,A -85,B 0,C 180,E1 -1966.49,E2 -1966.49} C_VEL
LIN {X 0,Y 580.801,Z 450.92,A -85,B 0,C 180,E1 -1967.752,E2 -1967.752} C_VEL
LIN {X 0,Y 580.756,Z 464.227,A -85,B 0,C 180,E1 -1968.062,E2 -1968.062} C_VEL
LIN {X 0,Y 580.648,Z 476.285,A -85,B 0,C 180,E1 -1968.48,E2 -1968.48} C_VEL
LIN {X 0,Y 580.578,Z 487.755,A -85,B 0,C 180,E1 -1969.009,E2 -1969.009} C_VEL
LIN {X 0,Y 580.42,Z 499.525,A -85,B 0,C 180,E1 -1969.712,E2 -1969.712} C_VEL
LIN {X 0,Y 580.345,Z 510.026,A -85,B 0,C 180,E1 -1970.503,E2 -1970.503} C_VEL
LIN {X 0,Y 580.273,Z 518.654,A -85,B 0,C 180,E1 -1971.292,E2 -1971.292} C_VEL
LIN {X 0,Y 580.222,Z 527.965,A -85,B 0,C 180,E1 -1972.343,E2 -1972.343} C_VEL
LIN {X 0,Y 580.171,Z 535.346,A -85,B 0,C 180,E1 -1973.377,E2 -1973.377} C_VEL
LIN {X 0,Y 580.139,Z 541.452,A -85,B 0,C 180,E1 -1974.438,E2 -1974.438} C_VEL
LIN {X 0,Y 580.108,Z 546.198,A -85,B 0,C 180,E1 -1975.483,E2 -1975.483} C_VEL
LIN {X 0,Y 580.124,Z 549.826,A -85,B 0,C 180,E1 -1976.527,E2 -1976.527} C_VEL
LIN {X 0,Y 580.043,Z 551.701,A -85,B 0,C 180,E1 -1977.222,E2 -1977.222} C_VEL
LIN {X 0,Y 580.038,Z 553.124,A -85,B 0,C 180,E1 -1977.917,E2 -1977.917} C_VEL
LIN {X 0,Y 580.041,Z 554.761,A -85,B 0,C 180,E1 -1979.306,E2 -1979.306} C_VEL
LIN {X 0,Y 580.038,Z 554.996,A -85,B 0,C 180,E1 -1980,E2 -1980} C_VEL
LIN {X 0,Y 580.04,Z 554.808,A -85,B 0,C 180,E1 -1980.694,E2 -1980.694} C_VEL
LIN {X 0,Y 580.037,Z 553.282,A -85,B 0,C 180,E1 -1982.083,E2 -1982.083} C_VEL
LIN {X 0,Y 580.044,Z 551.907,A -85,B 0,C 180,E1 -1982.778,E2 -1982.778} C_VEL
LIN {X 0,Y 580.11,Z 549.041,A -85,B 0,C 180,E1 -1983.821,E2 -1983.821} C_VEL
LIN {X 0,Y 580.054,Z 545.141,A -85,B 0,C 180,E1 -1984.865,E2 -1984.865} C_VEL
LIN {X 0,Y 580.161,Z 540.081,A -85,B 0,C 180,E1 -1985.91,E2 -1985.91} C_VEL
LIN {X 0,Y 580.158,Z 533.748,A -85,B 0,C 180,E1 -1986.958,E2 -1986.958} C_VEL
LIN {X 0,Y 580.241,Z 525.872,A -85,B 0,C 180,E1 -1988.007,E2 -1988.007} C_VEL
LIN {X 0,Y 580.298,Z 517.791,A -85,B 0,C 180,E1 -1988.883,E2 -1988.883} C_VEL
LIN {X 0,Y 580.361,Z 507.914,A -85,B 0,C 180,E1 -1989.761,E2 -1989.761} C_VEL
LIN {X 0,Y 580.504,Z 496.9,A -85,B 0,C 180,E1 -1990.551,E2 -1990.551} C_VEL
LIN {X 0,Y 580.57,Z 486.045,A -85,B 0,C 180,E1 -1991.168,E2 -1991.168} C_VEL
LIN {X 0,Y 580.65,Z 474.103,A -85,B 0,C 180,E1 -1991.697,E2 -1991.697} C_VEL
LIN {X 0,Y 580.775,Z 461.065,A -85,B 0,C 180,E1 -1992.115,E2 -1992.115} C_VEL
LIN {X 0,Y 580.862,Z 448.135,A -85,B 0,C 180,E1 -1992.379,E2 -1992.379} C_VEL
LIN {X 0,Y 580.929,Z 401.345,A -85,B 0,C 180,E1 -1992.966,E2 -1992.966} C_VEL
LIN {X 0,Y 580.251,Z 395.54,A -85,B 0,C 180,E1 -1993.054,E2 -1993.054} C_VEL
LIN {X 0,Y 574.683,Z 376.856,A -85,B 0,C 180,E1 -1993.417,E2 -1993.417} C_VEL
LIN {X 0,Y 574.045,Z 371.05,A -85,B 0,C 180,E1 -1993.505,E2 -1993.505} C_VEL
LIN {X 0,Y 573.886,Z 349.07,A -85,B 0,C 180,E1 -1993.786,E2 -1993.786} C_VEL
LIN {X 0,Y 573.23,Z 345.264,A -85,B 0,C 180,E1 -1993.877,E2 -1993.877} C_VEL
LIN {X 0,Y 573.268,Z 335.075,A -85,B 0,C 180,E1 -1996.012,E2 -1996.012} C_VEL
LIN {X 0,Y 573.221,Z 335.078,A -85,B 0,C 180,E1 -1998.589,E2 -1998.589} C_VEL
LIN {X 0,Y 573.256,Z 335.082,A -85,B 0,C 180,E1 -2001.291,E2 -2001.291} C_VEL
LIN {X 0,Y 573.234,Z 335.077,A -85,B 0,C 180,E1 -2003.865,E2 -2003.865} C_VEL
LIN {X 0,Y 573.241,Z 335.075,A -85,B 0,C 180,E1 -2006.492,E2 -2006.492} C_VEL
LIN {X 0,Y 573.241,Z 335.076,A -85,B 0,C 180,E1 -2008.564,E2 -2008.564} C_VEL
LIN {X 0,Y 573.23,Z 335.083,A -85,B 0,C 180,E1 -2010.993,E2 -2010.993} C_VEL
LIN {X 0,Y 573.267,Z 335.076,A -85,B 0,C 180,E1 -2013.524,E2 -2013.524} C_VEL
LIN {X 0,Y 573.218,Z 335.077,A -85,B 0,C 180,E1 -2016.051,E2 -2016.051} C_VEL
LIN {X 0,Y 573.247,Z 335.077,A -85,B 0,C 180,E1 -2018.701,E2 -2018.701} C_VEL
LIN {X 0,Y 573.248,Z 335.076,A -85,B 0,C 180,E1 -2021.594,E2 -2021.594} C_VEL
LIN {X 0,Y 573.24,Z 335.075,A -85,B 0,C 180,E1 -2024.333,E2 -2024.333} C_VEL
LIN {X 0,Y 573.244,Z 335.079,A -85,B 0,C 180,E1 -2027.358,E2 -2027.358} C_VEL
LIN {X 0,Y 573.257,Z 335.076,A -85,B 0,C 180,E1 -2030.567,E2 -2030.567} C_VEL
LIN {X 0,Y 573.257,Z 335.081,A -85,B 0,C 180,E1 -2033.077,E2 -2033.077} C_VEL
LIN {X 0,Y 573.276,Z 335.071,A -85,B 0,C 180,E1 -2035.671,E2 -2035.671} C_VEL
LIN {X 0,Y 573.252,Z 335.074,A -85,B 0,C 180,E1 -2038.185,E2 -2038.185} C_VEL
LIN {X 0,Y 573.27,Z 335.077,A -85,B 0,C 180,E1 -2040.634,E2 -2040.634} C_VEL
LIN {X 0,Y 573.242,Z 335.075,A -85,B 0,C 180,E1 -2043.507,E2 -2043.507} C_VEL
LIN {X 0,Y 573.236,Z 335.076,A -85,B 0,C 180,E1 -2046.134,E2 -2046.134} C_VEL
LIN {X 0,Y 573.254,Z 335.077,A -85,B 0,C 180,E1 -2049.173,E2 -2049.173} C_VEL
LIN {X 0,Y 573.234,Z 335.076,A -85,B 0,C 180,E1 -2051.411,E2 -2051.411} C_VEL
LIN {X 0,Y 573.252,Z 335.073,A -85,B 0,C 180,E1 -2053.621,E2 -2053.621} C_VEL
LIN {X 0,Y 573.278,Z 335.07,A -85,B 0,C 180,E1 -2055.806,E2 -2055.806} C_VEL
LIN {X 0,Y 573.267,Z 335.08,A -85,B 0,C 180,E1 -2058.744,E2 -2058.744} C_VEL
LIN {X 0,Y 573.287,Z 335.069,A -85,B 0,C 180,E1 -2061.54,E2 -2061.54} C_VEL
LIN {X 0,Y 573.303,Z 335.073,A -85,B 0,C 180,E1 -2064.371,E2 -2064.371} C_VEL
LIN {X 0,Y 573.315,Z 335.066,A -85,B 0,C 180,E1 -2067.892,E2 -2067.892} C_VEL
LIN {X 0,Y 573.339,Z 335.069,A -85,B 0,C 180,E1 -2070.702,E2 -2070.702} C_VEL
LIN {X 0,Y 573.312,Z 335.071,A -85,B 0,C 180,E1 -2072.81,E2 -2072.81} C_VEL
LIN {X 0,Y 573.299,Z 335.067,A -85,B 0,C 180,E1 -2075.627,E2 -2075.627} C_VEL
LIN {X 0,Y 573.292,Z 335.077,A -85,B 0,C 180,E1 -2078.458,E2 -2078.458} C_VEL
LIN {X 0,Y 573.273,Z 335.07,A -85,B 0,C 180,E1 -2081.311,E2 -2081.311} C_VEL
LIN {X 0,Y 573.282,Z 335.078,A -85,B 0,C 180,E1 -2084.424,E2 -2084.424} C_VEL
LIN {X 0,Y 573.26,Z 335.072,A -85,B 0,C 180,E1 -2087.111,E2 -2087.111} C_VEL
LIN {X 0,Y 573.254,Z 335.079,A -85,B 0,C 180,E1 -2090.076,E2 -2090.076} C_VEL
LIN {X 0,Y 573.233,Z 335.076,A -85,B 0,C 180,E1 -2093.098,E2 -2093.098} C_VEL
LIN {X 0,Y 573.254,Z 335.073,A -85,B 0,C 180,E1 -2095.409,E2 -2095.409} C_VEL
LIN {X 0,Y 573.263,Z 335.078,A -85,B 0,C 180,E1 -2098.031,E2 -2098.031} C_VEL
LIN {X 0,Y 573.242,Z 335.075,A -85,B 0,C 180,E1 -2100.884,E2 -2100.884} C_VEL
LIN {X 0,Y 573.285,Z 335.07,A -85,B 0,C 180,E1 -2103.527,E2 -2103.527} C_VEL
LIN {X 0,Y 573.258,Z 335.081,A -85,B 0,C 180,E1 -2106.047,E2 -2106.047} C_VEL
LIN {X 0,Y 573.247,Z 335.075,A -85,B 0,C 180,E1 -2108.7,E2 -2108.7} C_VEL
LIN {X 0,Y 573.249,Z 335.076,A -85,B 0,C 180,E1 -2111.595,E2 -2111.595} C_VEL
LIN {X 0,Y 573.233,Z 335.08,A -85,B 0,C 180,E1 -2114.332,E2 -2114.332} C_VEL
LIN {X 0,Y 573.255,Z 335.074,A -85,B 0,C 180,E1 -2117.355,E2 -2117.355} C_VEL
LIN {X 0,Y 573.244,Z 335.077,A -85,B 0,C 180,E1 -2120.393,E2 -2120.393} C_VEL
LIN {X 0,Y 573.25,Z 335.073,A -85,B 0,C 180,E1 -2123.077,E2 -2123.077} C_VEL
LIN {X 0,Y 573.267,Z 335.077,A -85,B 0,C 180,E1 -2125.671,E2 -2125.671} C_VEL
LIN {X 0,Y 573.244,Z 335.079,A -85,B 0,C 180,E1 -2128.185,E2 -2128.185} C_VEL
LIN {X 0,Y 573.262,Z 335.072,A -85,B 0,C 180,E1 -2130.634,E2 -2130.634} C_VEL
LIN {X 0,Y 573.264,Z 335.076,A -85,B 0,C 180,E1 -2133.499,E2 -2133.499} C_VEL
LIN {X 0,Y 573.226,Z 335.08,A -85,B 0,C 180,E1 -2136.134,E2 -2136.134} C_VEL
LIN {X 0,Y 573.254,Z 335.074,A -85,B 0,C 180,E1 -2139.174,E2 -2139.174} C_VEL
LIN {X 0,Y 573.231,Z 335.08,A -85,B 0,C 180,E1 -2141.412,E2 -2141.412} C_VEL
LIN {X 0,Y 573.252,Z 335.081,A -85,B 0,C 180,E1 -2143.622,E2 -2143.622} C_VEL
LIN {X 0,Y 573.23,Z 335.075,A -85,B 0,C 180,E1 -2146.529,E2 -2146.529} C_VEL
LIN {X 0,Y 573.274,Z 335.07,A -85,B 0,C 180,E1 -2148.734,E2 -2148.734} C_VEL
LIN {X 0,Y 573.299,Z 335.076,A -85,B 0,C 180,E1 -2151.541,E2 -2151.541} C_VEL
LIN {X 0,Y 573.284,Z 335.069,A -85,B 0,C 180,E1 -2154.372,E2 -2154.372} C_VEL
LIN {X 0,Y 573.301,Z 335.071,A -85,B 0,C 180,E1 -2157.892,E2 -2157.892} C_VEL
LIN {X 0,Y 573.329,Z 335.063,A -85,B 0,C 180,E1 -2160.702,E2 -2160.702} C_VEL
LIN {X 0,Y 573.234,Z 335.085,A -85,B 0,C 180,E1 -2163.515,E2 -2163.515} C_VEL
LIN {X 0,Y 573.284,Z 335.076,A -85,B 0,C 180,E1 -2165.628,E2 -2165.628} C_VEL
LIN {X 0,Y 573.283,Z 335.069,A -85,B 0,C 180,E1 -2168.46,E2 -2168.46} C_VEL
LIN {X 0,Y 573.29,Z 335.076,A -85,B 0,C 180,E1 -2171.312,E2 -2171.312} C_VEL
LIN {X 0,Y 573.272,Z 335.07,A -85,B 0,C 180,E1 -2174.425,E2 -2174.425} C_VEL
LIN {X 0,Y 573.252,Z 335.079,A -85,B 0,C 180,E1 -2177.112,E2 -2177.112} C_VEL
LIN {X 0,Y 573.249,Z 335.073,A -85,B 0,C 180,E1 -2180.077,E2 -2180.077} C_VEL
LIN {X 0,Y 573.232,Z 335.075,A -85,B 0,C 180,E1 -2182.338,E2 -2182.338} C_VEL
LIN {X 0,Y 573.249,Z 335.08,A -85,B 0,C 180,E1 -2185.41,E2 -2185.41} C_VEL
LIN {X 0,Y 573.257,Z 335.072,A -85,B 0,C 180,E1 -2188.032,E2 -2188.032} C_VEL
LIN {X 0,Y 573.233,Z 335.08,A -85,B 0,C 180,E1 -2190.885,E2 -2190.885} C_VEL
LIN {X 0,Y 573.281,Z 335.073,A -85,B 0,C 180,E1 -2193.529,E2 -2193.529} C_VEL
LIN {X 0,Y 573.254,Z 335.072,A -85,B 0,C 180,E1 -2196.049,E2 -2196.049} C_VEL
LIN {X 0,Y 573.245,Z 335.077,A -85,B 0,C 180,E1 -2198.702,E2 -2198.702} C_VEL
LIN {X 0,Y 573.26,Z 335.074,A -85,B 0,C 180,E1 -2201.598,E2 -2201.598} C_VEL
LIN {X 0,Y 573.234,Z 335.076,A -85,B 0,C 180,E1 -2204.334,E2 -2204.334} C_VEL
LIN {X 0,Y 573.239,Z 335.079,A -85,B 0,C 180,E1 -2207.359,E2 -2207.359} C_VEL
LIN {X 0,Y 573.246,Z 335.075,A -85,B 0,C 180,E1 -2210.394,E2 -2210.394} C_VEL
LIN {X 0,Y 573.254,Z 335.08,A -85,B 0,C 180,E1 -2213.079,E2 -2213.079} C_VEL
LIN {X 0,Y 573.272,Z 335.071,A -85,B 0,C 180,E1 -2215.673,E2 -2215.673} C_VEL
LIN {X 0,Y 573.248,Z 335.074,A -85,B 0,C 180,E1 -2218.186,E2 -2218.186} C_VEL
LIN {X 0,Y 573.268,Z 335.078,A -85,B 0,C 180,E1 -2220.636,E2 -2220.636} C_VEL
LIN {X 0,Y 573.269,Z 335.075,A -85,B 0,C 180,E1 -2223.502,E2 -2223.502} C_VEL
LIN {X 0,Y 573.254,Z 335.102,A -85,B 0,C 180,E1 -2224.927,E2 -2224.927} C_VEL
LIN {X 0,Y 574.313,Z 341.469,A -85,B 0,C 180,E1 -2225.8,E2 -2225.8} C_VEL
LIN {X 0,Y 574.073,Z 362.219,A -85,B 0,C 180,E1 -2228.501,E2 -2228.501} C_VEL
LIN {X 0,Y 573.834,Z 383.387,A -85,B 0,C 180,E1 -2231.248,E2 -2231.248} C_VEL
LIN {X 0,Y 573.582,Z 406.347,A -85,B 0,C 180,E1 -2234.18,E2 -2234.18} C_VEL
LIN {X 0,Y 573.444,Z 421.953,A -85,B 0,C 180,E1 -2236.152,E2 -2236.152} C_VEL
LIN {X 0,Y 574.092,Z 426.794,A -85,B 0,C 180,E1 -2236.235,E2 -2236.235} C_VEL
LIN {X 0,Y 573.881,Z 530.994,A -85,B 0,C 180,E1 -2237.558,E2 -2237.558} C_VEL
LIN {X 0,Y 573.777,Z 544.25,A -85,B 0,C 180,E1 -2237.87,E2 -2237.87} C_VEL
LIN {X 0,Y 573.686,Z 557.175,A -85,B 0,C 180,E1 -2238.326,E2 -2238.326} C_VEL
LIN {X 0,Y 573.593,Z 568.644,A -85,B 0,C 180,E1 -2238.874,E2 -2238.874} C_VEL
LIN {X 0,Y 573.434,Z 580.215,A -85,B 0,C 180,E1 -2239.586,E2 -2239.586} C_VEL
LIN {X 0,Y 573.327,Z 590.611,A -85,B 0,C 180,E1 -2240.386,E2 -2240.386} C_VEL
LIN {X 0,Y 573.24,Z 599.121,A -85,B 0,C 180,E1 -2241.185,E2 -2241.185} C_VEL
LIN {X 0,Y 573.16,Z 606.968,A -85,B 0,C 180,E1 -2242.072,E2 -2242.072} C_VEL
LIN {X 0,Y 573.073,Z 614.585,A -85,B 0,C 180,E1 -2243.127,E2 -2243.127} C_VEL
LIN {X 0,Y 573.07,Z 621.684,A -85,B 0,C 180,E1 -2244.371,E2 -2244.371} C_VEL
LIN {X 0,Y 573.028,Z 626.375,A -85,B 0,C 180,E1 -2245.428,E2 -2245.428} C_VEL
LIN {X 0,Y 573.022,Z 629.96,A -85,B 0,C 180,E1 -2246.485,E2 -2246.485} C_VEL
LIN {X 0,Y 572.959,Z 631.81,A -85,B 0,C 180,E1 -2247.189,E2 -2247.189} C_VEL
LIN {X 0,Y 572.938,Z 633.2,A -85,B 0,C 180,E1 -2247.892,E2 -2247.892} C_VEL
LIN {X 0,Y 572.941,Z 634.785,A -85,B 0,C 180,E1 -2249.298,E2 -2249.298} C_VEL
LIN {X 0,Y 572.938,Z 635,A -85,B 0,C 180,E1 -2250.001,E2 -2250.001} C_VEL
LIN {X 0,Y 572.946,Z 634.185,A -85,B 0,C 180,E1 -2251.407,E2 -2251.407} C_VEL
LIN {X 0,Y 572.938,Z 633.198,A -85,B 0,C 180,E1 -2252.11,E2 -2252.11} C_VEL
LIN {X 0,Y 572.959,Z 631.808,A -85,B 0,C 180,E1 -2252.813,E2 -2252.813} C_VEL
LIN {X 0,Y 573.014,Z 628.893,A -85,B 0,C 180,E1 -2253.869,E2 -2253.869} C_VEL
LIN {X 0,Y 572.963,Z 624.946,A -85,B 0,C 180,E1 -2254.926,E2 -2254.926} C_VEL
LIN {X 0,Y 573.064,Z 618.872,A -85,B 0,C 180,E1 -2256.161,E2 -2256.161} C_VEL
LIN {X 0,Y 573.12,Z 612.232,A -85,B 0,C 180,E1 -2257.222,E2 -2257.222} C_VEL
LIN {X 0,Y 573.199,Z 603.984,A -85,B 0,C 180,E1 -2258.284,E2 -2258.284} C_VEL
LIN {X 0,Y 573.286,Z 595.53,A -85,B 0,C 180,E1 -2259.171,E2 -2259.171} C_VEL
LIN {X 0,Y 573.421,Z 585.088,A -85,B 0,C 180,E1 -2260.059,E2 -2260.059} C_VEL
LIN {X 0,Y 573.528,Z 573.344,A -85,B 0,C 180,E1 -2260.859,E2 -2260.859} C_VEL
LIN {X 0,Y 573.655,Z 562.266,A -85,B 0,C 180,E1 -2261.448,E2 -2261.448} C_VEL
LIN {X 0,Y 573.759,Z 549.151,A -85,B 0,C 180,E1 -2261.975,E2 -2261.975} C_VEL
LIN {X 0,Y 573.869,Z 536.489,A -85,B 0,C 180,E1 -2262.331,E2 -2262.331} C_VEL
LIN {X 0,Y 573.923,Z 523.251,A -85,B 0,C 180,E1 -2262.555,E2 -2262.555} C_VEL
LIN {X 0,Y 574.019,Z 425.993,A -85,B 0,C 180,E1 -2263.777,E2 -2263.777} C_VEL
LIN {X 0,Y 573.446,Z 421.94,A -85,B 0,C 180,E1 -2263.85,E2 -2263.85} C_VEL
LIN {X 0,Y 573.663,Z 399.171,A -85,B 0,C 180,E1 -2266.731,E2 -2266.731} C_VEL
LIN {X 0,Y 573.874,Z 378.061,A -85,B 0,C 180,E1 -2269.44,E2 -2269.44} C_VEL
LIN {X 0,Y 574.142,Z 357.543,A -85,B 0,C 180,E1 -2272.112,E2 -2272.112} C_VEL
LIN {X 0,Y 574.287,Z 341.279,A -85,B 0,C 180,E1 -2274.203,E2 -2274.203} C_VEL
LIN {X 0,Y 573.247,Z 335.083,A -85,B 0,C 180,E1 -2275.034,E2 -2275.034} C_VEL
LIN {X 0,Y 573.277,Z 335.073,A -85,B 0,C 180,E1 -2277.766,E2 -2277.766} C_VEL
LIN {X 0,Y 573.255,Z 335.073,A -85,B 0,C 180,E1 -2280.176,E2 -2280.176} C_VEL
LIN {X 0,Y 573.26,Z 335.076,A -85,B 0,C 180,E1 -2282.645,E2 -2282.645} C_VEL
LIN {X 0,Y 573.246,Z 335.083,A -85,B 0,C 180,E1 -2285.186,E2 -2285.186} C_VEL
LIN {X 0,Y 573.241,Z 335.075,A -85,B 0,C 180,E1 -2287.808,E2 -2287.808} C_VEL
LIN {X 0,Y 573.25,Z 335.076,A -85,B 0,C 180,E1 -2290.525,E2 -2290.525} C_VEL
LIN {X 0,Y 573.244,Z 335.079,A -85,B 0,C 180,E1 -2293.359,E2 -2293.359} C_VEL
LIN {X 0,Y 573.25,Z 335.074,A -85,B 0,C 180,E1 -2296.331,E2 -2296.331} C_VEL
LIN {X 0,Y 573.245,Z 335.077,A -85,B 0,C 180,E1 -2298.544,E2 -2298.544} C_VEL
LIN {X 0,Y 573.248,Z 335.078,A -85,B 0,C 180,E1 -2301.299,E2 -2301.299} C_VEL
LIN {X 0,Y 573.218,Z 335.077,A -85,B 0,C 180,E1 -2304.019,E2 -2304.019} C_VEL
LIN {X 0,Y 573.275,Z 335.074,A -85,B 0,C 180,E1 -2306.518,E2 -2306.518} C_VEL
LIN {X 0,Y 573.234,Z 335.081,A -85,B 0,C 180,E1 -2309.118,E2 -2309.118} C_VEL
LIN {X 0,Y 573.256,Z 335.073,A -85,B 0,C 180,E1 -2311.971,E2 -2311.971} C_VEL
LIN {X 0,Y 573.258,Z 335.079,A -85,B 0,C 180,E1 -2314.59,E2 -2314.59} C_VEL
LIN {X 0,Y 573.241,Z 335.075,A -85,B 0,C 180,E1 -2317.662,E2 -2317.662} C_VEL
LIN {X 0,Y 573.271,Z 335.08,A -85,B 0,C 180,E1 -2320.67,E2 -2320.67} C_VEL
LIN {X 0,Y 573.262,Z 335.075,A -85,B 0,C 180,E1 -2323.622,E2 -2323.622} C_VEL
LIN {X 0,Y 573.256,Z 335.231,A -85,B 0,C 180,E1 -2324.124,E2 -2324.124} C_VEL
LIN {X 0,Y 573.208,Z 345.375,A -85,B 0,C 180,E1 -2326.235,E2 -2326.235} C_VEL
LIN {X 0,Y 574.056,Z 350.297,A -85,B 0,C 180,E1 -2326.324,E2 -2326.324} C_VEL
LIN {X 0,Y 573.886,Z 450.948,A -85,B 0,C 180,E1 -2327.602,E2 -2327.602} C_VEL
LIN {X 0,Y 573.815,Z 464.255,A -85,B 0,C 180,E1 -2327.915,E2 -2327.915} C_VEL
LIN {X 0,Y 573.702,Z 475.183,A -85,B 0,C 180,E1 -2328.294,E2 -2328.294} C_VEL
